// TIA Portal V17 export
// export: Created 2025-03-05T08:00:17.191262Z, ExportSetting WithDefaults, DisplayName Totally Integrated Automation Portal, DisplayVersion V17 Update 8, DisplayName TIA Portal Openness, DisplayVersion V17 Update 8, DisplayName TIA Portal Version Control Interface, DisplayVersion V17, DisplayName SINAMICS Startdrive Advanced, DisplayVersion V17 SP2, DisplayName SINAMICS Startdrive G110M, G120, G120C, G120D, G120P, G115D, DisplayVersion V17 SP2, DisplayName SINAMICS Startdrive G130, G150, S120, S150, SINAMICS MV, S210, DisplayVersion V17 SP2, DisplayName STEP 7 Professional, DisplayVersion V17 Update 8, DisplayName SINUMERIK ONE STEP 7 Toolbox, DisplayVersion V17 Update 12, DisplayName SINUMERIK 840D sl STEP 7 Toolbox, DisplayVersion V17 Update 12, DisplayName STEP 7 Safety, DisplayVersion V17 Update 6, DisplayName WinCC Advanced, DisplayVersion V17 Update 8
FUNCTION_BLOCK "FB33_SAFETY_POSITIONS"   // FB33, LAD
{ S7_Optimized_Access := 'FALSE' }
VERSION : 0.1
// stored: AutoNumber true, IsIECCheckEnabled false, SetENOAutomatically false, UDAEnableTagReadback false
   VAR_INPUT
      MEAS_SYS_1_ACTIVE_REFERENCED : Bool;   // MEASURING SYSTEM 1 ACTIVE AND REFERENCED
      MEAS_SYS_2_ACTIVE_REFERENCED : Bool;   // MEASURING SYSTEM 2 ACTIVE AND REFERENCED
      AXIS_POS : Real;   // AXIS POSITION
   END_VAR
   VAR DB_SPECIFIC
      AX_POS_0_DEGREES : Struct   // AXIS POSITION 0 DEGREES
         TOLERANCE : Real := 0.005;   // TOLERANCE
         POSITION_0_TOLERANCE_PLUS : Real;   // POSITION TOLERANCE PLUS
         POSITION_0_TOLERANCE_MINUS : Real;   // POSITION TOLERANCE MINUS
         POSITION_360_TOLERANCE_PLUS : Real;   // POSITION TOLERANCE PLUS
         POSITION_360_TOLERANCE_MINUS : Real;   // POSITION TOLERANCE MINUS
         IN_POSITION : Bool;   // AXIS POSITION 0 DEGREES
      END_STRUCT;
      AX_POS_90_DEGREES : Struct   // AXIS POSITION 90 DEGREES
         TOLERANCE : Real := 0.005;   // TOLERANCE
         POSITION_TOLERANCE_PLUS : Real;   // POSITION TOLERANCE PLUS
         POSITION_TOLERANCE_MINUS : Real;   // POSITION TOLERANCE MINUS
         IN_POSITION : Bool;   // AXIS POSITION 90 DEGREES
      END_STRUCT;
      AX_POS_180_DEGREES : Struct   // AXIS POSITION 180 DEGREES
         TOLERANCE : Real := 0.005;   // TOLERANCE
         POSITION_TOLERANCE_PLUS : Real;   // POSITION TOLERANCE PLUS
         POSITION_TOLERANCE_MINUS : Real;   // POSITION TOLERANCE MINUS
         IN_POSITION : Bool;   // AXIS POSITION 180 DEGREES
      END_STRUCT;
      AX_POS_270_DEGREES : Struct   // AXIS POSITION 270 DEGREES
         TOLERANCE : Real := 0.005;   // TOLERANCE
         POSITION_TOLERANCE_PLUS : Real;   // POSITION TOLERANCE PLUS
         POSITION_TOLERANCE_MINUS : Real;   // POSITION TOLERANCE MINUS
         IN_POSITION : Bool;   // AXIS POSITION 270 DEGREES
      END_STRUCT;
      AX_POS_MINUS_90_DEGREES : Bool;   // AXIS POSITION MINUS 90 DEGREES
      AX_POS_MINUS_180_DEGREES : Bool;   // AXIS POSITION MINUS 180 DEGREES
      AX_POS_MINUS_270_DEGREES : Bool;   // AXIS POSITION MINUS 270 DEGREES
      SAFETY_POSITION_1 : Struct   // HOME POSITION
         HMI_POSITION : Real := 1.1;   // HMI POSITION
         TOLERANCE_PLUS : Real := 0.01;   // TOLERANCE PLUS
         TOLERANCE_MINUS : Real := 0.01;   // TOLERANCE MINUS
         POSITION_TOLERANCE_PLUS : Real;   // POSITION TOLERANCE PLUS
         POSITION_TOLERANCE_MINUS : Real;   // POSITION TOLERANCE MINUS
         IN_POSITION : Bool;   // HOME POSITION
         GREATER_TOLERANCE_PLUS : Bool;   // GREATER THAN TOLERANCE PLUS
         GREATER_TOLERANCE_MINUS : Bool;   // GREATER TOLERANCE MINUS
         LOWER_TOLERANCE_PLUS : Bool;   // LOWER TOLERANCE PLUS
         LOWER_TOLERANCE_MINUS : Bool;   // LOWER TOLERANCE MINUS
      END_STRUCT;
      SAFETY_POSITION_2 : Struct   // CLEAR FIXTURE AXIS
         HMI_POSITION : Real := 1.1;   // HMI POSITION
         TOLERANCE_PLUS : Real := 0.01;   // TOLERANCE PLUS
         TOLERANCE_MINUS : Real := 0.01;   // TOLERANCE MINUS
         POSITION_TOLERANCE_PLUS : Real;   // POSITION TOLERANCE PLUS
         POSITION_TOLERANCE_MINUS : Real;   // POSITION TOLERANCE MINUS
         IN_POSITION : Bool;   // IN POSITION
         GREATER_TOLERANCE_PLUS : Bool;   // GREATER TOLERANCE PLUS
         GREATER_TOLERANCE_MINUS : Bool;   // CLEAR FIXTURE AXIS
         LOWER_TOLERANCE_PLUS : Bool;   // LOWER TOLERANCE PLUS
         LOWER_TOLERANCE_MINUS : Bool;   // LOWER TOLERANCE MINUS
      END_STRUCT;
      SAFETY_POSITION_3 : Struct   // TOOL CHANGE POSITION
         HMI_POSITION : Real := 1.1;   // HMI POSITION
         TOLERANCE_PLUS : Real := 0.01;   // TOLERANCE
         TOLERANCE_MINUS : Real := 0.01;   // TOLERANCE MINUS
         POSITION_TOLERANCE_PLUS : Real;   // POSITION TOLERANCE PLUS
         POSITION_TOLERANCE_MINUS : Real;   // POSITION TOLERANCE MINUS
         IN_POSITION : Bool;   // TOOL CHANGE POSITION
         GREATER_TOLERANCE_PLUS : Bool;   // GREATER TOLERANCE PLUS
         GREATER_TOLERANCE_MINUS : Bool;   // GREATER TOLERANCE MINUS
         LOWER_TOLERANCE_PLUS : Bool;   // LOWER TOLERANCE PLUS
         LOWER_TOLERANCE_MINUS : Bool;   // LOWER TOLERANCE MINUS
      END_STRUCT;
      SAFETY_POSITION_4 : Struct   // RETURNED
         HMI_POSITION : Real := 1.1;   // HMI POSITION
         TOLERANCE_PLUS : Real := 0.01;   // TOLERANCE PLUS
         TOLERANCE_MINUS : Real := 0.01;   // TOLERANCE MINUS
         POSITION_TOLERANCE_PLUS : Real;   // POSITION TOLERANCE PLUS
         POSITION_TOLERANCE_MINUS : Real;   // POSITION TOLERANCE MINUS
         IN_POSITION : Bool;   // RETURNED
         GREATER_TOLERANCE_PLUS : Bool;   // GREATER TOLERANCE PLUS
         GREATER_TOLERANCE_MINUS : Bool;   // GREATER TOLERANCE MINUS
         LOWER_TOLERANCE_PLUS : Bool;   // LOWER TOLERANCE PLUS
         LOWER_TOLERANCE_MINUS : Bool;   // LOWER TOLERANCE MINUS
      END_STRUCT;
      SAFETY_POSITION_5 : Struct   // ADVANCED
         HMI_POSITION : Real := 1.1;   // HMI POSITION
         TOLERANCE_PLUS : Real := 0.01;   // TOLERANCE_PLUS
         TOLERANCE_MINUS : Real := 0.01;   // TOLERANCE MINUS
         POSITION_TOLERANCE_PLUS : Real;   // POSITION TOLERANCE PLUS
         POSITION_TOLERANCE_MINUS : Real;   // POSITION TOLERANCE MINUS
         IN_POSITION : Bool;   // ADVANCED
         GREATER_TOLERANCE_PLUS : Bool;   // GREATER TOLERANCE PLUS
         GREATER_TOLERANCE_MINUS : Bool;   // GREATER TOLERANCE MINUS
         LOWER_TOLERANCE_PLUS : Bool;   // LOWER TOLERANCE PLUS
         LOWER_TOLERANCE_MINUS : Bool;   // LOWER TOLERANCE MINUS
      END_STRUCT;
      SAFETY_POSITION_6 : Struct
         HMI_POSITION : Real := 1.1;   // HMI POSITION
         TOLERANCE_PLUS : Real := 0.01;   // TOLERANCE PLUS
         TOLERANCE_MINUS : Real := 0.01;   // TOLERANCE MINUS
         POSITION_TOLERANCE_PLUS : Real;   // POSITION TOLERANCE PLUS
         POSITION_TOLERANCE_MINUS : Real;   // POSITION TOLERANCE MINUS
         IN_POSITION : Bool;   // IN POSITION
         GREATER_TOLERANCE_PLUS : Bool;   // GREATER TOLERANCE PLUS
         GREATER_TOLERANCE_MINUS : Bool;   // GREATER TOLERANCE MINUS
         LOWER_TOLERANCE_PLUS : Bool;   // LOWER TOLERANCE PLUS
         LOWER_TOLERANCE_MINUS : Bool;   // LOWER TOLERANCE MINUS
      END_STRUCT;
      SAFETY_POSITION_7 : Struct
         HMI_POSITION : Real := 1.1;   // HMI POSITION
         TOLERANCE_PLUS : Real := 0.01;   // TOLERANCE PLUS
         TOLERANCE_MINUS : Real := 0.01;   // TOLERANCE MINUS
         POSITION_TOLERANCE_PLUS : Real;   // POSITION TOLERANCE PLUS
         POSITION_TOLERANCE_MINUS : Real;   // POSITION TOLERANCE MINUS
         IN_POSITION : Bool;   // IN POSITION
         GREATER_TOLERANCE_PLUS : Bool;   // GREATER TOLERANCE PLUS
         GREATER_TOLERANCE_MINUS : Bool;   // GREATER TOLERANCE MINUS
         LOWER_TOLERANCE_PLUS : Bool;   // LOWER TOLERANCE PLUS
         LOWER_TOLERANCE_MINUS : Bool;   // LOWER TOLERANCE MINUS
      END_STRUCT;
      SAFETY_POSITION_8 : Struct
         HMI_POSITION : Real := 1.1;   // HMI POSITION
         TOLERANCE_PLUS : Real := 0.01;   // TOLERANCE PLUS
         TOLERANCE_MINUS : Real := 0.01;   // TOLERANCE MINUS
         POSITION_TOLERANCE_PLUS : Real;   // POSITION TOLERANCE PLUS
         POSITION_TOLERANCE_MINUS : Real;   // POSITION TOLERANCE MINUS
         IN_POSITION : Bool;   // IN POSITION
         GREATER_TOLERANCE_PLUS : Bool;   // GREATER TOLERANCE PLUS
         GREATER_TOLERANCE_MINUS : Bool;   // GREATER TOLERANCE MINUS
         LOWER_TOLERANCE_PLUS : Bool;   // LOWER TOLERANCE PLUS
         LOWER_TOLERANCE_MINUS : Bool;   // LOWER TOLERANCE MINUS
      END_STRUCT;
      SAFETY_POSITION_9 : Struct
         HMI_POSITION : Real := 1.1;   // HMI POSITION
         TOLERANCE_PLUS : Real := 0.01;   // TOLERANCE PLUS
         TOLERANCE_MINUS : Real := 0.01;   // TOLERANCE MINUS
         POSITION_TOLERANCE_PLUS : Real;   // POSITION TOLERANCE PLUS
         POSITION_TOLERANCE_MINUS : Real;   // POSITION TOLERANCE MINUS
         IN_POSITION : Bool;   // IN POSITION
         GREATER_TOLERANCE_PLUS : Bool;   // GREATER TOLERANCE PLUS
         GREATER_TOLERANCE_MINUS : Bool;   // GREATER TOLERANCE MINUS
         LOWER_TOLERANCE_PLUS : Bool;   // LOWER TOLERANCE PLUS
         LOWER_TOLERANCE_MINUS : Bool;   // LOWER TOLERANCE MINUS
      END_STRUCT;
      SAFETY_POSITION_10 : Struct
         HMI_POSITION : Real := 1.1;   // HMI POSITION
         TOLERANCE_PLUS : Real := 0.01;   // TOLERANCE PLUS
         TOLERANCE_MINUS : Real := 0.01;   // TOLERANCE MINUS
         POSITION_TOLERANCE_PLUS : Real;   // POSITION TOLERANCE PLUS
         POSITION_TOLERANCE_MINUS : Real;   // POSITION TOLERANCE MINUS
         IN_POSITION : Bool;   // IN POSITION
         GREATER_TOLERANCE_PLUS : Bool;   // GREATER TOLERANCE PLUS
         GREATER_TOLERANCE_MINUS : Bool;   // GREATER TOLERANCE MINUS
         LOWER_TOLERANCE_PLUS : Bool;   // LOWER TOLERANCE PLUS
         LOWER_TOLERANCE_MINUS : Bool;   // LOWER TOLERANCE MINUS
      END_STRUCT;
   END_VAR
   VAR_TEMP   // added for the SCL form of the ladder/FBD networks
      _w1 : Bool;
      _w2 : Bool;
   END_VAR
BEGIN

REGION Network 1: AXIS POSITION 0 DEGREES
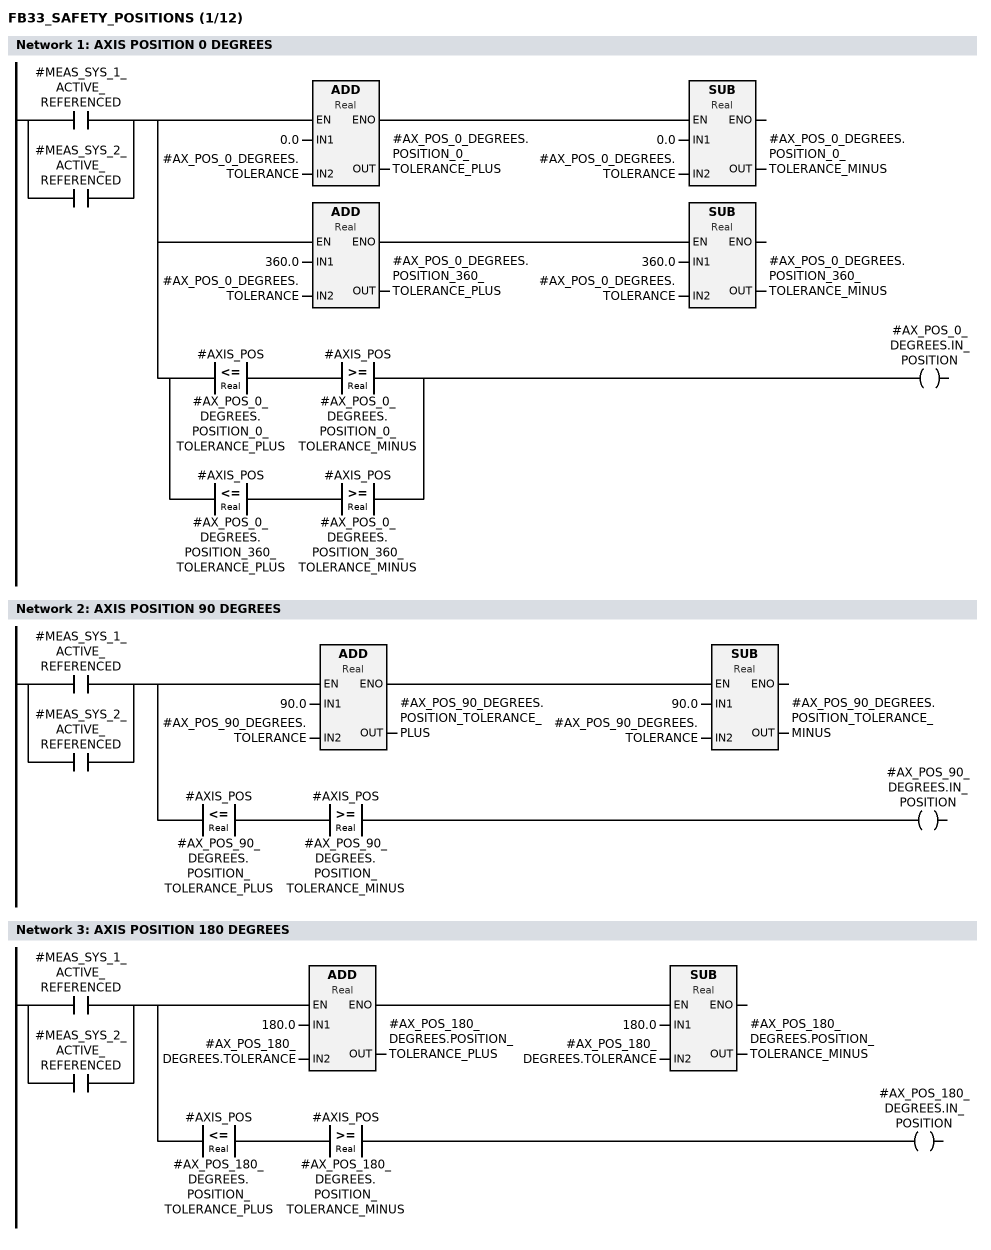
   RUNG wire#powerrail
      Contact( #MEAS_SYS_1_ACTIVE_REFERENCED )
      wire#w1
      { S7_Templates := "SrcType := Real"; S7_GenerateENO := "TRUE" } Add(in1 := 0.0, in2 := #AX_POS_0_DEGREES.TOLERANCE, out => #AX_POS_0_DEGREES.POSITION_0_TOLERANCE_PLUS)
      { S7_Templates := "SrcType := Real"; S7_GenerateENO := "TRUE" } Sub(in1 := 0.0, in2 := #AX_POS_0_DEGREES.TOLERANCE, out => #AX_POS_0_DEGREES.POSITION_0_TOLERANCE_MINUS)
   END_RUNG
   RUNG wire#powerrail
      Contact( #MEAS_SYS_2_ACTIVE_REFERENCED )
   END_RUNG wire#w1
   RUNG wire#w1
      { S7_Templates := "SrcType := Real"; S7_GenerateENO := "TRUE" } Add(in1 := 360.0, in2 := #AX_POS_0_DEGREES.TOLERANCE, out => #AX_POS_0_DEGREES.POSITION_360_TOLERANCE_PLUS)
      { S7_Templates := "SrcType := Real"; S7_GenerateENO := "TRUE" } Sub(in1 := 360.0, in2 := #AX_POS_0_DEGREES.TOLERANCE, out => #AX_POS_0_DEGREES.POSITION_360_TOLERANCE_MINUS)
   END_RUNG
   RUNG wire#w1
      { S7_Templates := "SrcType := Real" } LE_Contact(in1 := #AXIS_POS, in2 := #AX_POS_0_DEGREES.POSITION_0_TOLERANCE_PLUS)
      { S7_Templates := "SrcType := Real" } GE_Contact(in1 := #AXIS_POS, in2 := #AX_POS_0_DEGREES.POSITION_0_TOLERANCE_MINUS)
      wire#w2
      Coil( #AX_POS_0_DEGREES.IN_POSITION )
   END_RUNG
   RUNG wire#w1
      { S7_Templates := "SrcType := Real" } LE_Contact(in1 := #AXIS_POS, in2 := #AX_POS_0_DEGREES.POSITION_360_TOLERANCE_PLUS)
      { S7_Templates := "SrcType := Real" } GE_Contact(in1 := #AXIS_POS, in2 := #AX_POS_0_DEGREES.POSITION_360_TOLERANCE_MINUS)
   END_RUNG wire#w2
   // the same network as SCL:
   // ENO of a box is taken as its EN; it also drops when the box reports an error
   #_w1 := #MEAS_SYS_1_ACTIVE_REFERENCED OR #MEAS_SYS_2_ACTIVE_REFERENCED;
   IF #_w1 THEN
       #AX_POS_0_DEGREES.POSITION_0_TOLERANCE_PLUS := 0.0 + #AX_POS_0_DEGREES.TOLERANCE;
       #AX_POS_0_DEGREES.POSITION_0_TOLERANCE_MINUS := 0.0 - #AX_POS_0_DEGREES.TOLERANCE;
       #AX_POS_0_DEGREES.POSITION_360_TOLERANCE_PLUS := 360.0 + #AX_POS_0_DEGREES.TOLERANCE;
       #AX_POS_0_DEGREES.POSITION_360_TOLERANCE_MINUS := 360.0 - #AX_POS_0_DEGREES.TOLERANCE;
   END_IF;
   #AX_POS_0_DEGREES.IN_POSITION := #_w1 AND (((#AXIS_POS <= #AX_POS_0_DEGREES.POSITION_0_TOLERANCE_PLUS) AND (#AXIS_POS >= #AX_POS_0_DEGREES.POSITION_0_TOLERANCE_MINUS)) OR ((#AXIS_POS <= #AX_POS_0_DEGREES.POSITION_360_TOLERANCE_PLUS) AND (#AXIS_POS >= #AX_POS_0_DEGREES.POSITION_360_TOLERANCE_MINUS)));
END_REGION

REGION Network 2: AXIS POSITION 90 DEGREES
   RUNG wire#powerrail
      Contact( #MEAS_SYS_1_ACTIVE_REFERENCED )
      wire#w1
      { S7_Templates := "SrcType := Real"; S7_GenerateENO := "TRUE" } Add(in1 := 90.0, in2 := #AX_POS_90_DEGREES.TOLERANCE, out => #AX_POS_90_DEGREES.POSITION_TOLERANCE_PLUS)
      { S7_Templates := "SrcType := Real"; S7_GenerateENO := "TRUE" } Sub(in1 := 90.0, in2 := #AX_POS_90_DEGREES.TOLERANCE, out => #AX_POS_90_DEGREES.POSITION_TOLERANCE_MINUS)
   END_RUNG
   RUNG wire#powerrail
      Contact( #MEAS_SYS_2_ACTIVE_REFERENCED )
   END_RUNG wire#w1
   RUNG wire#w1
      { S7_Templates := "SrcType := Real" } LE_Contact(in1 := #AXIS_POS, in2 := #AX_POS_90_DEGREES.POSITION_TOLERANCE_PLUS)
      { S7_Templates := "SrcType := Real" } GE_Contact(in1 := #AXIS_POS, in2 := #AX_POS_90_DEGREES.POSITION_TOLERANCE_MINUS)
      Coil( #AX_POS_90_DEGREES.IN_POSITION )
   END_RUNG
   // the same network as SCL:
   // ENO of a box is taken as its EN; it also drops when the box reports an error
   #_w1 := #MEAS_SYS_1_ACTIVE_REFERENCED OR #MEAS_SYS_2_ACTIVE_REFERENCED;
   IF #_w1 THEN
       #AX_POS_90_DEGREES.POSITION_TOLERANCE_PLUS := 90.0 + #AX_POS_90_DEGREES.TOLERANCE;
       #AX_POS_90_DEGREES.POSITION_TOLERANCE_MINUS := 90.0 - #AX_POS_90_DEGREES.TOLERANCE;
   END_IF;
   #AX_POS_90_DEGREES.IN_POSITION := #_w1 AND (#AXIS_POS <= #AX_POS_90_DEGREES.POSITION_TOLERANCE_PLUS) AND (#AXIS_POS >= #AX_POS_90_DEGREES.POSITION_TOLERANCE_MINUS);
END_REGION

REGION Network 3: AXIS POSITION 180 DEGREES
   RUNG wire#powerrail
      Contact( #MEAS_SYS_1_ACTIVE_REFERENCED )
      wire#w1
      { S7_Templates := "SrcType := Real"; S7_GenerateENO := "TRUE" } Add(in1 := 180.0, in2 := #AX_POS_180_DEGREES.TOLERANCE, out => #AX_POS_180_DEGREES.POSITION_TOLERANCE_PLUS)
      { S7_Templates := "SrcType := Real"; S7_GenerateENO := "TRUE" } Sub(in1 := 180.0, in2 := #AX_POS_180_DEGREES.TOLERANCE, out => #AX_POS_180_DEGREES.POSITION_TOLERANCE_MINUS)
   END_RUNG
   RUNG wire#powerrail
      Contact( #MEAS_SYS_2_ACTIVE_REFERENCED )
   END_RUNG wire#w1
   RUNG wire#w1
      { S7_Templates := "SrcType := Real" } LE_Contact(in1 := #AXIS_POS, in2 := #AX_POS_180_DEGREES.POSITION_TOLERANCE_PLUS)
      { S7_Templates := "SrcType := Real" } GE_Contact(in1 := #AXIS_POS, in2 := #AX_POS_180_DEGREES.POSITION_TOLERANCE_MINUS)
      Coil( #AX_POS_180_DEGREES.IN_POSITION )
   END_RUNG
   // the same network as SCL:
   // ENO of a box is taken as its EN; it also drops when the box reports an error
   #_w1 := #MEAS_SYS_1_ACTIVE_REFERENCED OR #MEAS_SYS_2_ACTIVE_REFERENCED;
   IF #_w1 THEN
       #AX_POS_180_DEGREES.POSITION_TOLERANCE_PLUS := 180.0 + #AX_POS_180_DEGREES.TOLERANCE;
       #AX_POS_180_DEGREES.POSITION_TOLERANCE_MINUS := 180.0 - #AX_POS_180_DEGREES.TOLERANCE;
   END_IF;
   #AX_POS_180_DEGREES.IN_POSITION := #_w1 AND (#AXIS_POS <= #AX_POS_180_DEGREES.POSITION_TOLERANCE_PLUS) AND (#AXIS_POS >= #AX_POS_180_DEGREES.POSITION_TOLERANCE_MINUS);
END_REGION

REGION Network 4: AXIS POSITION 270 DEGREES
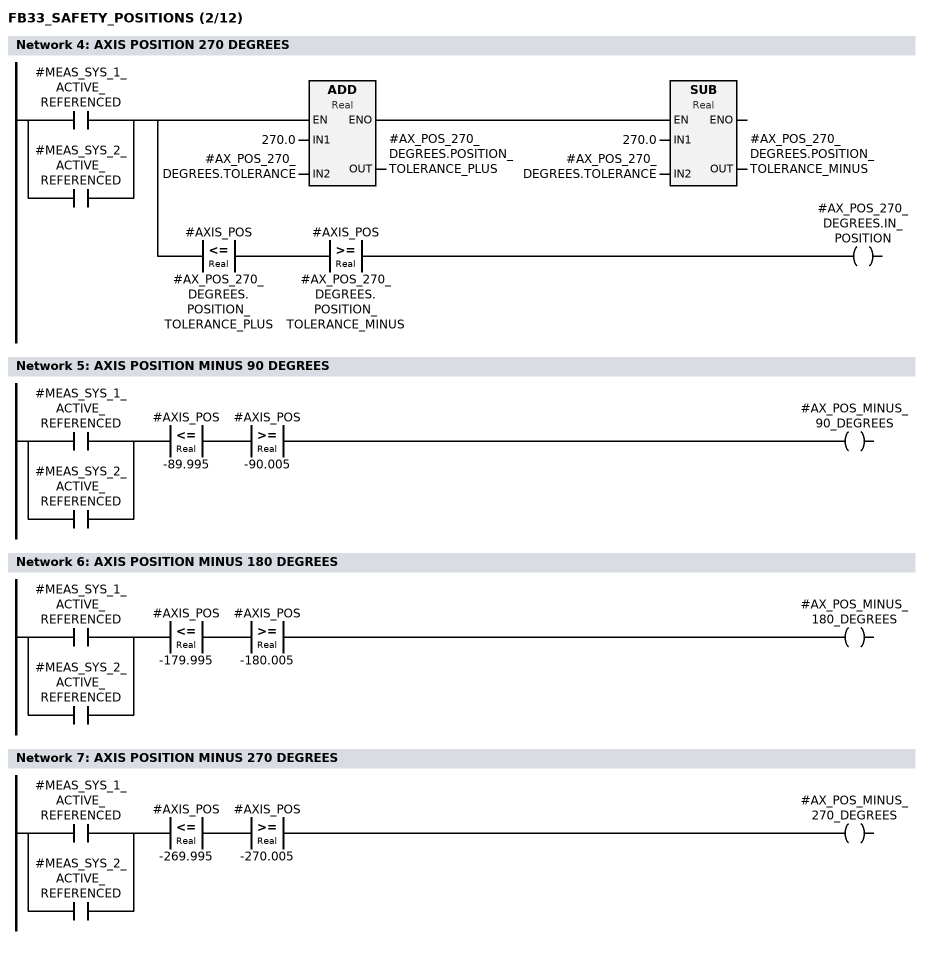
   RUNG wire#powerrail
      Contact( #MEAS_SYS_1_ACTIVE_REFERENCED )
      wire#w1
      { S7_Templates := "SrcType := Real"; S7_GenerateENO := "TRUE" } Add(in1 := 270.0, in2 := #AX_POS_270_DEGREES.TOLERANCE, out => #AX_POS_270_DEGREES.POSITION_TOLERANCE_PLUS)
      { S7_Templates := "SrcType := Real"; S7_GenerateENO := "TRUE" } Sub(in1 := 270.0, in2 := #AX_POS_270_DEGREES.TOLERANCE, out => #AX_POS_270_DEGREES.POSITION_TOLERANCE_MINUS)
   END_RUNG
   RUNG wire#powerrail
      Contact( #MEAS_SYS_2_ACTIVE_REFERENCED )
   END_RUNG wire#w1
   RUNG wire#w1
      { S7_Templates := "SrcType := Real" } LE_Contact(in1 := #AXIS_POS, in2 := #AX_POS_270_DEGREES.POSITION_TOLERANCE_PLUS)
      { S7_Templates := "SrcType := Real" } GE_Contact(in1 := #AXIS_POS, in2 := #AX_POS_270_DEGREES.POSITION_TOLERANCE_MINUS)
      Coil( #AX_POS_270_DEGREES.IN_POSITION )
   END_RUNG
   // the same network as SCL:
   // ENO of a box is taken as its EN; it also drops when the box reports an error
   #_w1 := #MEAS_SYS_1_ACTIVE_REFERENCED OR #MEAS_SYS_2_ACTIVE_REFERENCED;
   IF #_w1 THEN
       #AX_POS_270_DEGREES.POSITION_TOLERANCE_PLUS := 270.0 + #AX_POS_270_DEGREES.TOLERANCE;
       #AX_POS_270_DEGREES.POSITION_TOLERANCE_MINUS := 270.0 - #AX_POS_270_DEGREES.TOLERANCE;
   END_IF;
   #AX_POS_270_DEGREES.IN_POSITION := #_w1 AND (#AXIS_POS <= #AX_POS_270_DEGREES.POSITION_TOLERANCE_PLUS) AND (#AXIS_POS >= #AX_POS_270_DEGREES.POSITION_TOLERANCE_MINUS);
END_REGION

REGION Network 5: AXIS POSITION MINUS 90 DEGREES
   RUNG wire#powerrail
      Contact( #MEAS_SYS_1_ACTIVE_REFERENCED )
      wire#w1
      { S7_Templates := "SrcType := Real" } LE_Contact(in1 := #AXIS_POS, in2 := -89.995)
      { S7_Templates := "SrcType := Real" } GE_Contact(in1 := #AXIS_POS, in2 := -90.005)
      Coil( #AX_POS_MINUS_90_DEGREES )
   END_RUNG
   RUNG wire#powerrail
      Contact( #MEAS_SYS_2_ACTIVE_REFERENCED )
   END_RUNG wire#w1
   // the same network as SCL:
   #AX_POS_MINUS_90_DEGREES := (#MEAS_SYS_1_ACTIVE_REFERENCED OR #MEAS_SYS_2_ACTIVE_REFERENCED) AND (#AXIS_POS <= (-89.995)) AND (#AXIS_POS >= (-90.005));
END_REGION

REGION Network 6: AXIS POSITION MINUS 180 DEGREES
   RUNG wire#powerrail
      Contact( #MEAS_SYS_1_ACTIVE_REFERENCED )
      wire#w1
      { S7_Templates := "SrcType := Real" } LE_Contact(in1 := #AXIS_POS, in2 := -179.995)
      { S7_Templates := "SrcType := Real" } GE_Contact(in1 := #AXIS_POS, in2 := -180.005)
      Coil( #AX_POS_MINUS_180_DEGREES )
   END_RUNG
   RUNG wire#powerrail
      Contact( #MEAS_SYS_2_ACTIVE_REFERENCED )
   END_RUNG wire#w1
   // the same network as SCL:
   #AX_POS_MINUS_180_DEGREES := (#MEAS_SYS_1_ACTIVE_REFERENCED OR #MEAS_SYS_2_ACTIVE_REFERENCED) AND (#AXIS_POS <= (-179.995)) AND (#AXIS_POS >= (-180.005));
END_REGION

REGION Network 7: AXIS POSITION MINUS 270 DEGREES
   RUNG wire#powerrail
      Contact( #MEAS_SYS_1_ACTIVE_REFERENCED )
      wire#w1
      { S7_Templates := "SrcType := Real" } LE_Contact(in1 := #AXIS_POS, in2 := -269.995)
      { S7_Templates := "SrcType := Real" } GE_Contact(in1 := #AXIS_POS, in2 := -270.005)
      Coil( #AX_POS_MINUS_270_DEGREES )
   END_RUNG
   RUNG wire#powerrail
      Contact( #MEAS_SYS_2_ACTIVE_REFERENCED )
   END_RUNG wire#w1
   // the same network as SCL:
   #AX_POS_MINUS_270_DEGREES := (#MEAS_SYS_1_ACTIVE_REFERENCED OR #MEAS_SYS_2_ACTIVE_REFERENCED) AND (#AXIS_POS <= (-269.995)) AND (#AXIS_POS >= (-270.005));
END_REGION

REGION Network 8: SAFETY POSITION 1
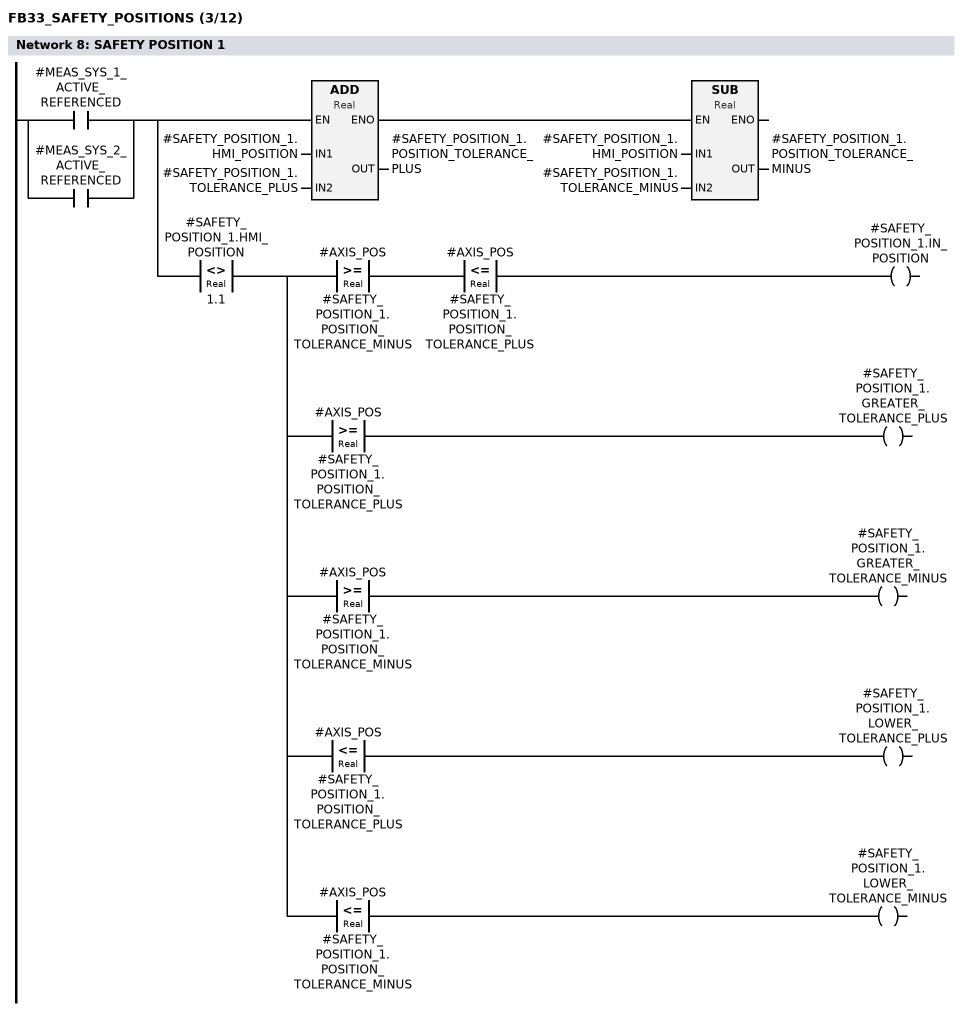
   RUNG wire#powerrail
      Contact( #MEAS_SYS_1_ACTIVE_REFERENCED )
      wire#w1
      { S7_Templates := "SrcType := Real"; S7_GenerateENO := "TRUE" } Add(in1 := #SAFETY_POSITION_1.HMI_POSITION, in2 := #SAFETY_POSITION_1.TOLERANCE_PLUS, out => #SAFETY_POSITION_1.POSITION_TOLERANCE_PLUS)
      { S7_Templates := "SrcType := Real"; S7_GenerateENO := "TRUE" } Sub(in1 := #SAFETY_POSITION_1.HMI_POSITION, in2 := #SAFETY_POSITION_1.TOLERANCE_MINUS, out => #SAFETY_POSITION_1.POSITION_TOLERANCE_MINUS)
   END_RUNG
   RUNG wire#powerrail
      Contact( #MEAS_SYS_2_ACTIVE_REFERENCED )
   END_RUNG wire#w1
   RUNG wire#w1
      { S7_Templates := "SrcType := Real" } NE_Contact(in1 := #SAFETY_POSITION_1.HMI_POSITION, in2 := 1.1)
      wire#w2
      { S7_Templates := "SrcType := Real" } GE_Contact(in1 := #AXIS_POS, in2 := #SAFETY_POSITION_1.POSITION_TOLERANCE_MINUS)
      { S7_Templates := "SrcType := Real" } LE_Contact(in1 := #AXIS_POS, in2 := #SAFETY_POSITION_1.POSITION_TOLERANCE_PLUS)
      Coil( #SAFETY_POSITION_1.IN_POSITION )
   END_RUNG
   RUNG wire#w2
      { S7_Templates := "SrcType := Real" } GE_Contact(in1 := #AXIS_POS, in2 := #SAFETY_POSITION_1.POSITION_TOLERANCE_PLUS)
      Coil( #SAFETY_POSITION_1.GREATER_TOLERANCE_PLUS )
   END_RUNG
   RUNG wire#w2
      { S7_Templates := "SrcType := Real" } GE_Contact(in1 := #AXIS_POS, in2 := #SAFETY_POSITION_1.POSITION_TOLERANCE_MINUS)
      Coil( #SAFETY_POSITION_1.GREATER_TOLERANCE_MINUS )
   END_RUNG
   RUNG wire#w2
      { S7_Templates := "SrcType := Real" } LE_Contact(in1 := #AXIS_POS, in2 := #SAFETY_POSITION_1.POSITION_TOLERANCE_PLUS)
      Coil( #SAFETY_POSITION_1.LOWER_TOLERANCE_PLUS )
   END_RUNG
   RUNG wire#w2
      { S7_Templates := "SrcType := Real" } LE_Contact(in1 := #AXIS_POS, in2 := #SAFETY_POSITION_1.POSITION_TOLERANCE_MINUS)
      Coil( #SAFETY_POSITION_1.LOWER_TOLERANCE_MINUS )
   END_RUNG
   // the same network as SCL:
   // ENO of a box is taken as its EN; it also drops when the box reports an error
   #_w1 := #MEAS_SYS_1_ACTIVE_REFERENCED OR #MEAS_SYS_2_ACTIVE_REFERENCED;
   IF #_w1 THEN
       #SAFETY_POSITION_1.POSITION_TOLERANCE_PLUS := #SAFETY_POSITION_1.HMI_POSITION + #SAFETY_POSITION_1.TOLERANCE_PLUS;
       #SAFETY_POSITION_1.POSITION_TOLERANCE_MINUS := #SAFETY_POSITION_1.HMI_POSITION - #SAFETY_POSITION_1.TOLERANCE_MINUS;
   END_IF;
   #_w2 := #_w1 AND (#SAFETY_POSITION_1.HMI_POSITION <> 1.1);
   #SAFETY_POSITION_1.IN_POSITION := #_w2 AND (#AXIS_POS >= #SAFETY_POSITION_1.POSITION_TOLERANCE_MINUS) AND (#AXIS_POS <= #SAFETY_POSITION_1.POSITION_TOLERANCE_PLUS);
   #SAFETY_POSITION_1.GREATER_TOLERANCE_PLUS := #_w2 AND (#AXIS_POS >= #SAFETY_POSITION_1.POSITION_TOLERANCE_PLUS);
   #SAFETY_POSITION_1.GREATER_TOLERANCE_MINUS := #_w2 AND (#AXIS_POS >= #SAFETY_POSITION_1.POSITION_TOLERANCE_MINUS);
   #SAFETY_POSITION_1.LOWER_TOLERANCE_PLUS := #_w2 AND (#AXIS_POS <= #SAFETY_POSITION_1.POSITION_TOLERANCE_PLUS);
   #SAFETY_POSITION_1.LOWER_TOLERANCE_MINUS := #_w2 AND (#AXIS_POS <= #SAFETY_POSITION_1.POSITION_TOLERANCE_MINUS);
END_REGION

REGION Network 9: SAFETY POSITION 2
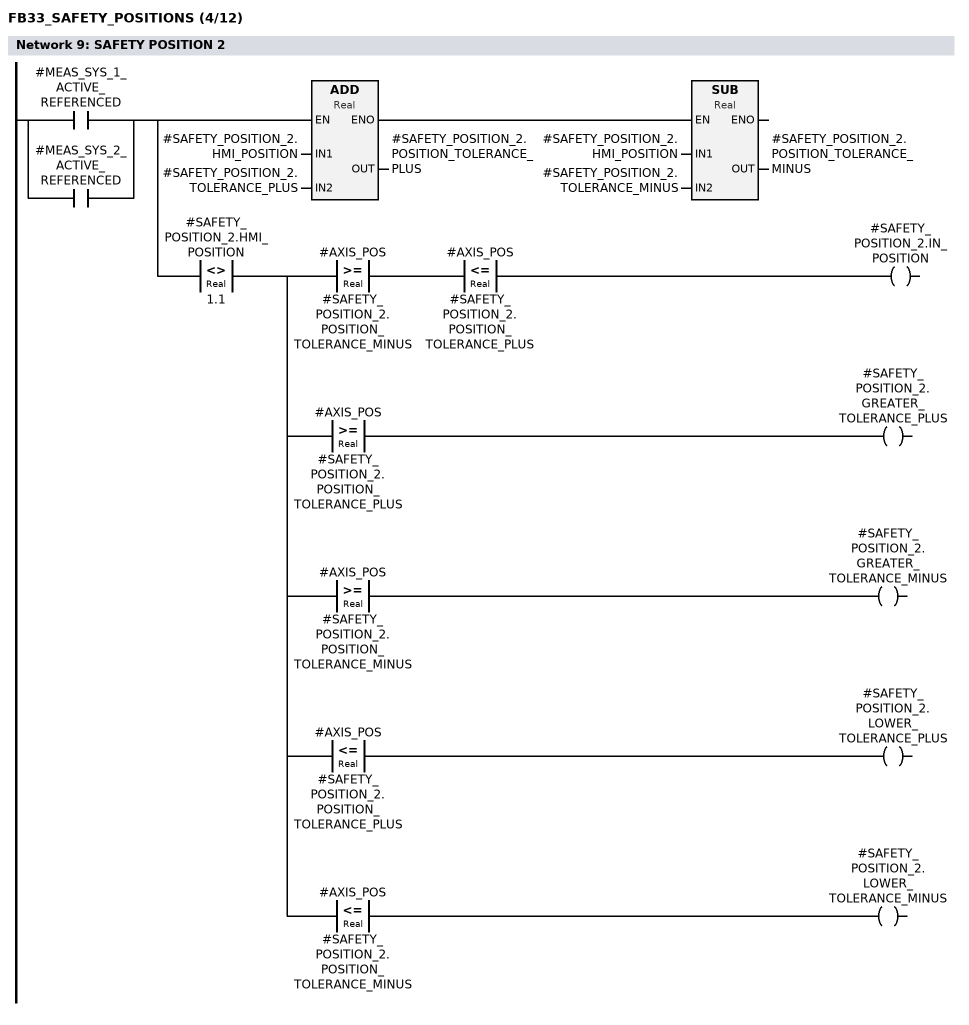
   RUNG wire#powerrail
      Contact( #MEAS_SYS_1_ACTIVE_REFERENCED )
      wire#w1
      { S7_Templates := "SrcType := Real"; S7_GenerateENO := "TRUE" } Add(in1 := #SAFETY_POSITION_2.HMI_POSITION, in2 := #SAFETY_POSITION_2.TOLERANCE_PLUS, out => #SAFETY_POSITION_2.POSITION_TOLERANCE_PLUS)
      { S7_Templates := "SrcType := Real"; S7_GenerateENO := "TRUE" } Sub(in1 := #SAFETY_POSITION_2.HMI_POSITION, in2 := #SAFETY_POSITION_2.TOLERANCE_MINUS, out => #SAFETY_POSITION_2.POSITION_TOLERANCE_MINUS)
   END_RUNG
   RUNG wire#powerrail
      Contact( #MEAS_SYS_2_ACTIVE_REFERENCED )
   END_RUNG wire#w1
   RUNG wire#w1
      { S7_Templates := "SrcType := Real" } NE_Contact(in1 := #SAFETY_POSITION_2.HMI_POSITION, in2 := 1.1)
      wire#w2
      { S7_Templates := "SrcType := Real" } GE_Contact(in1 := #AXIS_POS, in2 := #SAFETY_POSITION_2.POSITION_TOLERANCE_MINUS)
      { S7_Templates := "SrcType := Real" } LE_Contact(in1 := #AXIS_POS, in2 := #SAFETY_POSITION_2.POSITION_TOLERANCE_PLUS)
      Coil( #SAFETY_POSITION_2.IN_POSITION )
   END_RUNG
   RUNG wire#w2
      { S7_Templates := "SrcType := Real" } GE_Contact(in1 := #AXIS_POS, in2 := #SAFETY_POSITION_2.POSITION_TOLERANCE_PLUS)
      Coil( #SAFETY_POSITION_2.GREATER_TOLERANCE_PLUS )
   END_RUNG
   RUNG wire#w2
      { S7_Templates := "SrcType := Real" } GE_Contact(in1 := #AXIS_POS, in2 := #SAFETY_POSITION_2.POSITION_TOLERANCE_MINUS)
      Coil( #SAFETY_POSITION_2.GREATER_TOLERANCE_MINUS )
   END_RUNG
   RUNG wire#w2
      { S7_Templates := "SrcType := Real" } LE_Contact(in1 := #AXIS_POS, in2 := #SAFETY_POSITION_2.POSITION_TOLERANCE_PLUS)
      Coil( #SAFETY_POSITION_2.LOWER_TOLERANCE_PLUS )
   END_RUNG
   RUNG wire#w2
      { S7_Templates := "SrcType := Real" } LE_Contact(in1 := #AXIS_POS, in2 := #SAFETY_POSITION_2.POSITION_TOLERANCE_MINUS)
      Coil( #SAFETY_POSITION_2.LOWER_TOLERANCE_MINUS )
   END_RUNG
   // the same network as SCL:
   // ENO of a box is taken as its EN; it also drops when the box reports an error
   #_w1 := #MEAS_SYS_1_ACTIVE_REFERENCED OR #MEAS_SYS_2_ACTIVE_REFERENCED;
   IF #_w1 THEN
       #SAFETY_POSITION_2.POSITION_TOLERANCE_PLUS := #SAFETY_POSITION_2.HMI_POSITION + #SAFETY_POSITION_2.TOLERANCE_PLUS;
       #SAFETY_POSITION_2.POSITION_TOLERANCE_MINUS := #SAFETY_POSITION_2.HMI_POSITION - #SAFETY_POSITION_2.TOLERANCE_MINUS;
   END_IF;
   #_w2 := #_w1 AND (#SAFETY_POSITION_2.HMI_POSITION <> 1.1);
   #SAFETY_POSITION_2.IN_POSITION := #_w2 AND (#AXIS_POS >= #SAFETY_POSITION_2.POSITION_TOLERANCE_MINUS) AND (#AXIS_POS <= #SAFETY_POSITION_2.POSITION_TOLERANCE_PLUS);
   #SAFETY_POSITION_2.GREATER_TOLERANCE_PLUS := #_w2 AND (#AXIS_POS >= #SAFETY_POSITION_2.POSITION_TOLERANCE_PLUS);
   #SAFETY_POSITION_2.GREATER_TOLERANCE_MINUS := #_w2 AND (#AXIS_POS >= #SAFETY_POSITION_2.POSITION_TOLERANCE_MINUS);
   #SAFETY_POSITION_2.LOWER_TOLERANCE_PLUS := #_w2 AND (#AXIS_POS <= #SAFETY_POSITION_2.POSITION_TOLERANCE_PLUS);
   #SAFETY_POSITION_2.LOWER_TOLERANCE_MINUS := #_w2 AND (#AXIS_POS <= #SAFETY_POSITION_2.POSITION_TOLERANCE_MINUS);
END_REGION

REGION Network 10: SAFETY POSITION 3
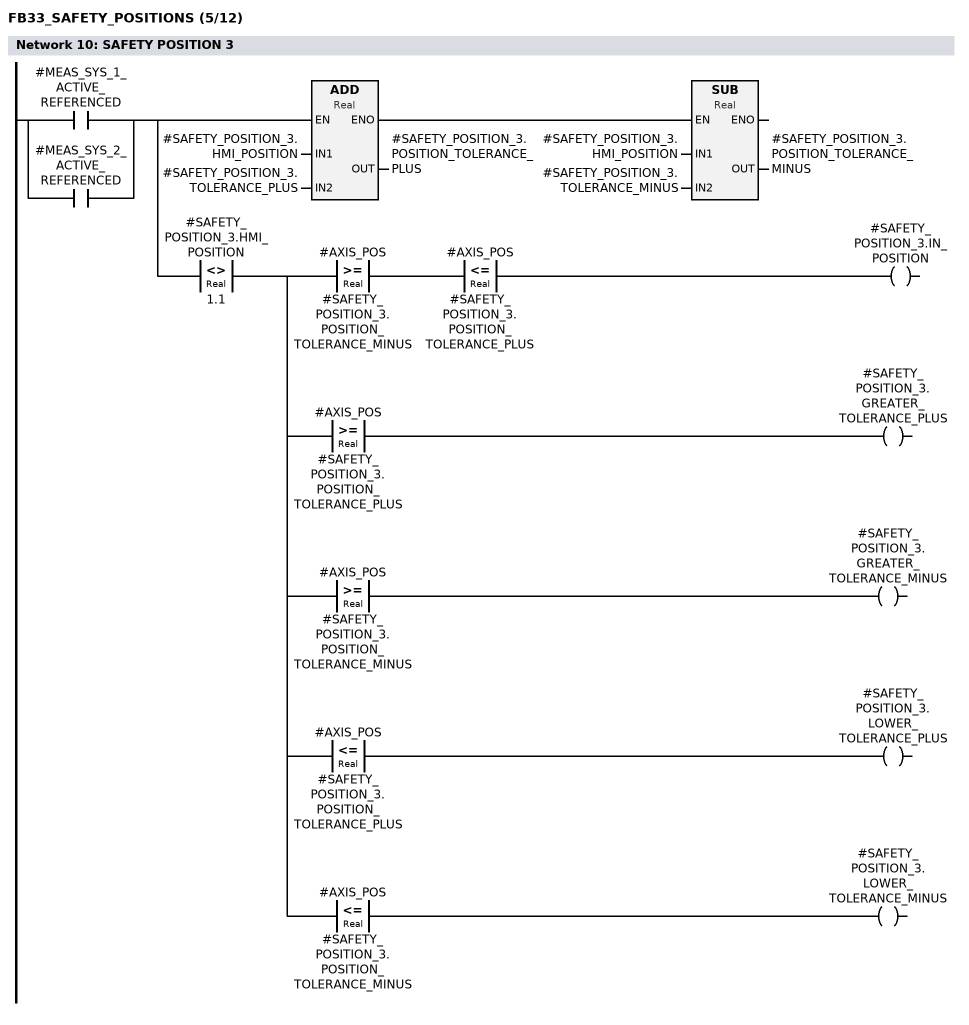
   RUNG wire#powerrail
      Contact( #MEAS_SYS_1_ACTIVE_REFERENCED )
      wire#w1
      { S7_Templates := "SrcType := Real"; S7_GenerateENO := "TRUE" } Add(in1 := #SAFETY_POSITION_3.HMI_POSITION, in2 := #SAFETY_POSITION_3.TOLERANCE_PLUS, out => #SAFETY_POSITION_3.POSITION_TOLERANCE_PLUS)
      { S7_Templates := "SrcType := Real"; S7_GenerateENO := "TRUE" } Sub(in1 := #SAFETY_POSITION_3.HMI_POSITION, in2 := #SAFETY_POSITION_3.TOLERANCE_MINUS, out => #SAFETY_POSITION_3.POSITION_TOLERANCE_MINUS)
   END_RUNG
   RUNG wire#powerrail
      Contact( #MEAS_SYS_2_ACTIVE_REFERENCED )
   END_RUNG wire#w1
   RUNG wire#w1
      { S7_Templates := "SrcType := Real" } NE_Contact(in1 := #SAFETY_POSITION_3.HMI_POSITION, in2 := 1.1)
      wire#w2
      { S7_Templates := "SrcType := Real" } GE_Contact(in1 := #AXIS_POS, in2 := #SAFETY_POSITION_3.POSITION_TOLERANCE_MINUS)
      { S7_Templates := "SrcType := Real" } LE_Contact(in1 := #AXIS_POS, in2 := #SAFETY_POSITION_3.POSITION_TOLERANCE_PLUS)
      Coil( #SAFETY_POSITION_3.IN_POSITION )
   END_RUNG
   RUNG wire#w2
      { S7_Templates := "SrcType := Real" } GE_Contact(in1 := #AXIS_POS, in2 := #SAFETY_POSITION_3.POSITION_TOLERANCE_PLUS)
      Coil( #SAFETY_POSITION_3.GREATER_TOLERANCE_PLUS )
   END_RUNG
   RUNG wire#w2
      { S7_Templates := "SrcType := Real" } GE_Contact(in1 := #AXIS_POS, in2 := #SAFETY_POSITION_3.POSITION_TOLERANCE_MINUS)
      Coil( #SAFETY_POSITION_3.GREATER_TOLERANCE_MINUS )
   END_RUNG
   RUNG wire#w2
      { S7_Templates := "SrcType := Real" } LE_Contact(in1 := #AXIS_POS, in2 := #SAFETY_POSITION_3.POSITION_TOLERANCE_PLUS)
      Coil( #SAFETY_POSITION_3.LOWER_TOLERANCE_PLUS )
   END_RUNG
   RUNG wire#w2
      { S7_Templates := "SrcType := Real" } LE_Contact(in1 := #AXIS_POS, in2 := #SAFETY_POSITION_3.POSITION_TOLERANCE_MINUS)
      Coil( #SAFETY_POSITION_3.LOWER_TOLERANCE_MINUS )
   END_RUNG
   // the same network as SCL:
   // ENO of a box is taken as its EN; it also drops when the box reports an error
   #_w1 := #MEAS_SYS_1_ACTIVE_REFERENCED OR #MEAS_SYS_2_ACTIVE_REFERENCED;
   IF #_w1 THEN
       #SAFETY_POSITION_3.POSITION_TOLERANCE_PLUS := #SAFETY_POSITION_3.HMI_POSITION + #SAFETY_POSITION_3.TOLERANCE_PLUS;
       #SAFETY_POSITION_3.POSITION_TOLERANCE_MINUS := #SAFETY_POSITION_3.HMI_POSITION - #SAFETY_POSITION_3.TOLERANCE_MINUS;
   END_IF;
   #_w2 := #_w1 AND (#SAFETY_POSITION_3.HMI_POSITION <> 1.1);
   #SAFETY_POSITION_3.IN_POSITION := #_w2 AND (#AXIS_POS >= #SAFETY_POSITION_3.POSITION_TOLERANCE_MINUS) AND (#AXIS_POS <= #SAFETY_POSITION_3.POSITION_TOLERANCE_PLUS);
   #SAFETY_POSITION_3.GREATER_TOLERANCE_PLUS := #_w2 AND (#AXIS_POS >= #SAFETY_POSITION_3.POSITION_TOLERANCE_PLUS);
   #SAFETY_POSITION_3.GREATER_TOLERANCE_MINUS := #_w2 AND (#AXIS_POS >= #SAFETY_POSITION_3.POSITION_TOLERANCE_MINUS);
   #SAFETY_POSITION_3.LOWER_TOLERANCE_PLUS := #_w2 AND (#AXIS_POS <= #SAFETY_POSITION_3.POSITION_TOLERANCE_PLUS);
   #SAFETY_POSITION_3.LOWER_TOLERANCE_MINUS := #_w2 AND (#AXIS_POS <= #SAFETY_POSITION_3.POSITION_TOLERANCE_MINUS);
END_REGION

REGION Network 11: SAFETY POSITION 4
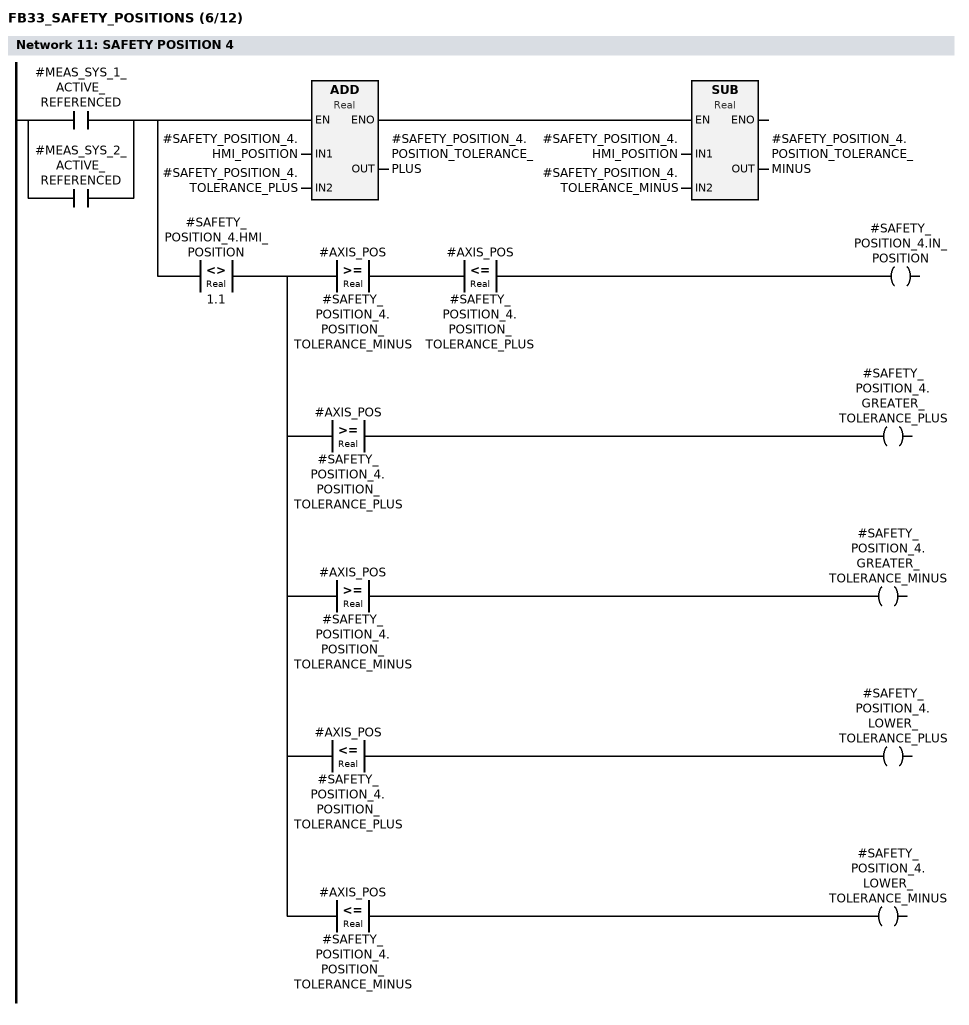
   RUNG wire#powerrail
      Contact( #MEAS_SYS_1_ACTIVE_REFERENCED )
      wire#w1
      { S7_Templates := "SrcType := Real"; S7_GenerateENO := "TRUE" } Add(in1 := #SAFETY_POSITION_4.HMI_POSITION, in2 := #SAFETY_POSITION_4.TOLERANCE_PLUS, out => #SAFETY_POSITION_4.POSITION_TOLERANCE_PLUS)
      { S7_Templates := "SrcType := Real"; S7_GenerateENO := "TRUE" } Sub(in1 := #SAFETY_POSITION_4.HMI_POSITION, in2 := #SAFETY_POSITION_4.TOLERANCE_MINUS, out => #SAFETY_POSITION_4.POSITION_TOLERANCE_MINUS)
   END_RUNG
   RUNG wire#powerrail
      Contact( #MEAS_SYS_2_ACTIVE_REFERENCED )
   END_RUNG wire#w1
   RUNG wire#w1
      { S7_Templates := "SrcType := Real" } NE_Contact(in1 := #SAFETY_POSITION_4.HMI_POSITION, in2 := 1.1)
      wire#w2
      { S7_Templates := "SrcType := Real" } GE_Contact(in1 := #AXIS_POS, in2 := #SAFETY_POSITION_4.POSITION_TOLERANCE_MINUS)
      { S7_Templates := "SrcType := Real" } LE_Contact(in1 := #AXIS_POS, in2 := #SAFETY_POSITION_4.POSITION_TOLERANCE_PLUS)
      Coil( #SAFETY_POSITION_4.IN_POSITION )
   END_RUNG
   RUNG wire#w2
      { S7_Templates := "SrcType := Real" } GE_Contact(in1 := #AXIS_POS, in2 := #SAFETY_POSITION_4.POSITION_TOLERANCE_PLUS)
      Coil( #SAFETY_POSITION_4.GREATER_TOLERANCE_PLUS )
   END_RUNG
   RUNG wire#w2
      { S7_Templates := "SrcType := Real" } GE_Contact(in1 := #AXIS_POS, in2 := #SAFETY_POSITION_4.POSITION_TOLERANCE_MINUS)
      Coil( #SAFETY_POSITION_4.GREATER_TOLERANCE_MINUS )
   END_RUNG
   RUNG wire#w2
      { S7_Templates := "SrcType := Real" } LE_Contact(in1 := #AXIS_POS, in2 := #SAFETY_POSITION_4.POSITION_TOLERANCE_PLUS)
      Coil( #SAFETY_POSITION_4.LOWER_TOLERANCE_PLUS )
   END_RUNG
   RUNG wire#w2
      { S7_Templates := "SrcType := Real" } LE_Contact(in1 := #AXIS_POS, in2 := #SAFETY_POSITION_4.POSITION_TOLERANCE_MINUS)
      Coil( #SAFETY_POSITION_4.LOWER_TOLERANCE_MINUS )
   END_RUNG
   // the same network as SCL:
   // ENO of a box is taken as its EN; it also drops when the box reports an error
   #_w1 := #MEAS_SYS_1_ACTIVE_REFERENCED OR #MEAS_SYS_2_ACTIVE_REFERENCED;
   IF #_w1 THEN
       #SAFETY_POSITION_4.POSITION_TOLERANCE_PLUS := #SAFETY_POSITION_4.HMI_POSITION + #SAFETY_POSITION_4.TOLERANCE_PLUS;
       #SAFETY_POSITION_4.POSITION_TOLERANCE_MINUS := #SAFETY_POSITION_4.HMI_POSITION - #SAFETY_POSITION_4.TOLERANCE_MINUS;
   END_IF;
   #_w2 := #_w1 AND (#SAFETY_POSITION_4.HMI_POSITION <> 1.1);
   #SAFETY_POSITION_4.IN_POSITION := #_w2 AND (#AXIS_POS >= #SAFETY_POSITION_4.POSITION_TOLERANCE_MINUS) AND (#AXIS_POS <= #SAFETY_POSITION_4.POSITION_TOLERANCE_PLUS);
   #SAFETY_POSITION_4.GREATER_TOLERANCE_PLUS := #_w2 AND (#AXIS_POS >= #SAFETY_POSITION_4.POSITION_TOLERANCE_PLUS);
   #SAFETY_POSITION_4.GREATER_TOLERANCE_MINUS := #_w2 AND (#AXIS_POS >= #SAFETY_POSITION_4.POSITION_TOLERANCE_MINUS);
   #SAFETY_POSITION_4.LOWER_TOLERANCE_PLUS := #_w2 AND (#AXIS_POS <= #SAFETY_POSITION_4.POSITION_TOLERANCE_PLUS);
   #SAFETY_POSITION_4.LOWER_TOLERANCE_MINUS := #_w2 AND (#AXIS_POS <= #SAFETY_POSITION_4.POSITION_TOLERANCE_MINUS);
END_REGION

REGION Network 12: SAFETY POSITION 5
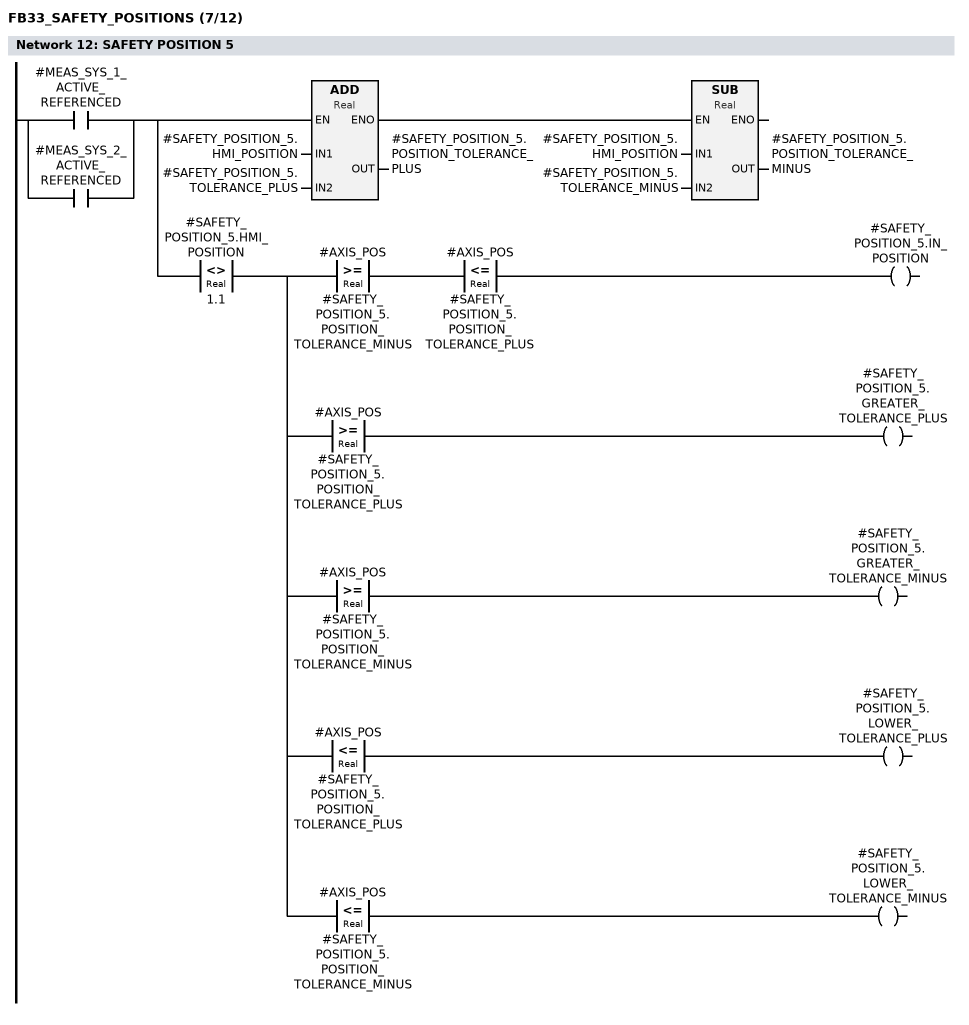
   RUNG wire#powerrail
      Contact( #MEAS_SYS_1_ACTIVE_REFERENCED )
      wire#w1
      { S7_Templates := "SrcType := Real"; S7_GenerateENO := "TRUE" } Add(in1 := #SAFETY_POSITION_5.HMI_POSITION, in2 := #SAFETY_POSITION_5.TOLERANCE_PLUS, out => #SAFETY_POSITION_5.POSITION_TOLERANCE_PLUS)
      { S7_Templates := "SrcType := Real"; S7_GenerateENO := "TRUE" } Sub(in1 := #SAFETY_POSITION_5.HMI_POSITION, in2 := #SAFETY_POSITION_5.TOLERANCE_MINUS, out => #SAFETY_POSITION_5.POSITION_TOLERANCE_MINUS)
   END_RUNG
   RUNG wire#powerrail
      Contact( #MEAS_SYS_2_ACTIVE_REFERENCED )
   END_RUNG wire#w1
   RUNG wire#w1
      { S7_Templates := "SrcType := Real" } NE_Contact(in1 := #SAFETY_POSITION_5.HMI_POSITION, in2 := 1.1)
      wire#w2
      { S7_Templates := "SrcType := Real" } GE_Contact(in1 := #AXIS_POS, in2 := #SAFETY_POSITION_5.POSITION_TOLERANCE_MINUS)
      { S7_Templates := "SrcType := Real" } LE_Contact(in1 := #AXIS_POS, in2 := #SAFETY_POSITION_5.POSITION_TOLERANCE_PLUS)
      Coil( #SAFETY_POSITION_5.IN_POSITION )
   END_RUNG
   RUNG wire#w2
      { S7_Templates := "SrcType := Real" } GE_Contact(in1 := #AXIS_POS, in2 := #SAFETY_POSITION_5.POSITION_TOLERANCE_PLUS)
      Coil( #SAFETY_POSITION_5.GREATER_TOLERANCE_PLUS )
   END_RUNG
   RUNG wire#w2
      { S7_Templates := "SrcType := Real" } GE_Contact(in1 := #AXIS_POS, in2 := #SAFETY_POSITION_5.POSITION_TOLERANCE_MINUS)
      Coil( #SAFETY_POSITION_5.GREATER_TOLERANCE_MINUS )
   END_RUNG
   RUNG wire#w2
      { S7_Templates := "SrcType := Real" } LE_Contact(in1 := #AXIS_POS, in2 := #SAFETY_POSITION_5.POSITION_TOLERANCE_PLUS)
      Coil( #SAFETY_POSITION_5.LOWER_TOLERANCE_PLUS )
   END_RUNG
   RUNG wire#w2
      { S7_Templates := "SrcType := Real" } LE_Contact(in1 := #AXIS_POS, in2 := #SAFETY_POSITION_5.POSITION_TOLERANCE_MINUS)
      Coil( #SAFETY_POSITION_5.LOWER_TOLERANCE_MINUS )
   END_RUNG
   // the same network as SCL:
   // ENO of a box is taken as its EN; it also drops when the box reports an error
   #_w1 := #MEAS_SYS_1_ACTIVE_REFERENCED OR #MEAS_SYS_2_ACTIVE_REFERENCED;
   IF #_w1 THEN
       #SAFETY_POSITION_5.POSITION_TOLERANCE_PLUS := #SAFETY_POSITION_5.HMI_POSITION + #SAFETY_POSITION_5.TOLERANCE_PLUS;
       #SAFETY_POSITION_5.POSITION_TOLERANCE_MINUS := #SAFETY_POSITION_5.HMI_POSITION - #SAFETY_POSITION_5.TOLERANCE_MINUS;
   END_IF;
   #_w2 := #_w1 AND (#SAFETY_POSITION_5.HMI_POSITION <> 1.1);
   #SAFETY_POSITION_5.IN_POSITION := #_w2 AND (#AXIS_POS >= #SAFETY_POSITION_5.POSITION_TOLERANCE_MINUS) AND (#AXIS_POS <= #SAFETY_POSITION_5.POSITION_TOLERANCE_PLUS);
   #SAFETY_POSITION_5.GREATER_TOLERANCE_PLUS := #_w2 AND (#AXIS_POS >= #SAFETY_POSITION_5.POSITION_TOLERANCE_PLUS);
   #SAFETY_POSITION_5.GREATER_TOLERANCE_MINUS := #_w2 AND (#AXIS_POS >= #SAFETY_POSITION_5.POSITION_TOLERANCE_MINUS);
   #SAFETY_POSITION_5.LOWER_TOLERANCE_PLUS := #_w2 AND (#AXIS_POS <= #SAFETY_POSITION_5.POSITION_TOLERANCE_PLUS);
   #SAFETY_POSITION_5.LOWER_TOLERANCE_MINUS := #_w2 AND (#AXIS_POS <= #SAFETY_POSITION_5.POSITION_TOLERANCE_MINUS);
END_REGION

REGION Network 13: SAFETY POSITION 6
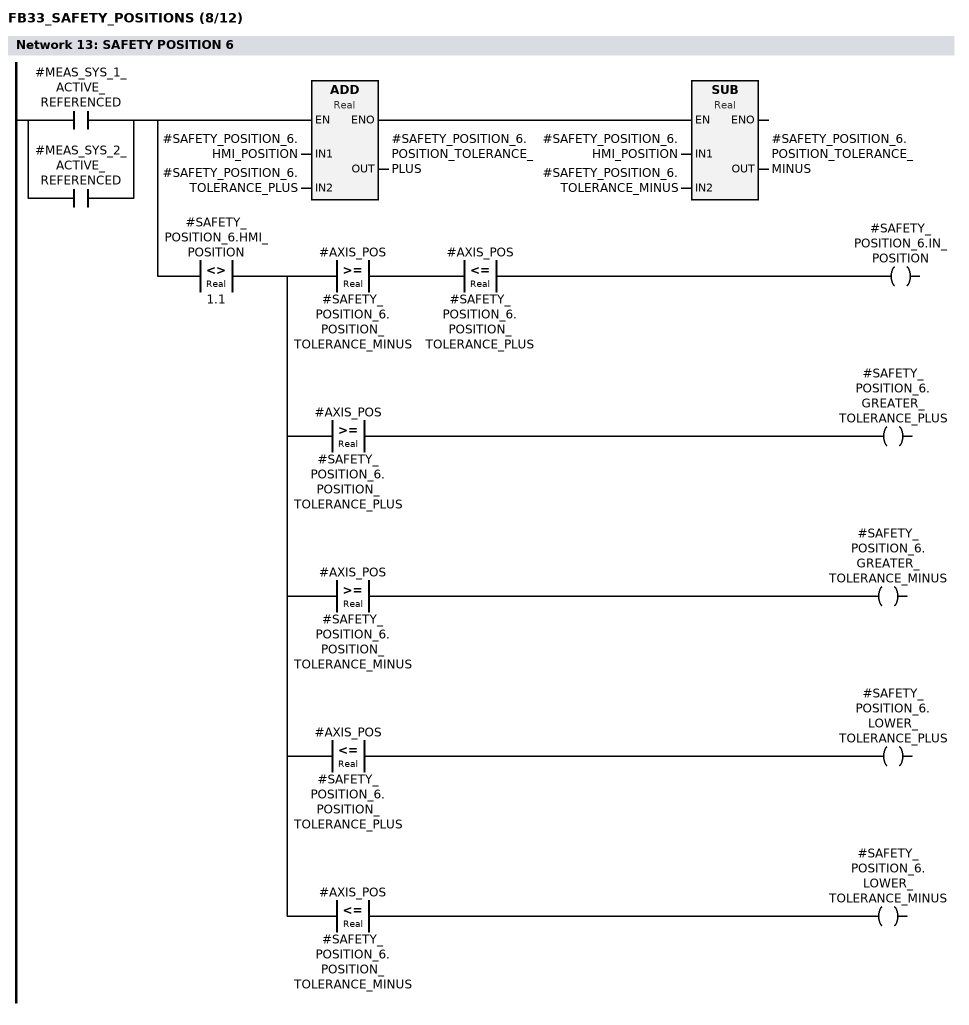
   RUNG wire#powerrail
      Contact( #MEAS_SYS_1_ACTIVE_REFERENCED )
      wire#w1
      { S7_Templates := "SrcType := Real"; S7_GenerateENO := "TRUE" } Add(in1 := #SAFETY_POSITION_6.HMI_POSITION, in2 := #SAFETY_POSITION_6.TOLERANCE_PLUS, out => #SAFETY_POSITION_6.POSITION_TOLERANCE_PLUS)
      { S7_Templates := "SrcType := Real"; S7_GenerateENO := "TRUE" } Sub(in1 := #SAFETY_POSITION_6.HMI_POSITION, in2 := #SAFETY_POSITION_6.TOLERANCE_MINUS, out => #SAFETY_POSITION_6.POSITION_TOLERANCE_MINUS)
   END_RUNG
   RUNG wire#powerrail
      Contact( #MEAS_SYS_2_ACTIVE_REFERENCED )
   END_RUNG wire#w1
   RUNG wire#w1
      { S7_Templates := "SrcType := Real" } NE_Contact(in1 := #SAFETY_POSITION_6.HMI_POSITION, in2 := 1.1)
      wire#w2
      { S7_Templates := "SrcType := Real" } GE_Contact(in1 := #AXIS_POS, in2 := #SAFETY_POSITION_6.POSITION_TOLERANCE_MINUS)
      { S7_Templates := "SrcType := Real" } LE_Contact(in1 := #AXIS_POS, in2 := #SAFETY_POSITION_6.POSITION_TOLERANCE_PLUS)
      Coil( #SAFETY_POSITION_6.IN_POSITION )
   END_RUNG
   RUNG wire#w2
      { S7_Templates := "SrcType := Real" } GE_Contact(in1 := #AXIS_POS, in2 := #SAFETY_POSITION_6.POSITION_TOLERANCE_PLUS)
      Coil( #SAFETY_POSITION_6.GREATER_TOLERANCE_PLUS )
   END_RUNG
   RUNG wire#w2
      { S7_Templates := "SrcType := Real" } GE_Contact(in1 := #AXIS_POS, in2 := #SAFETY_POSITION_6.POSITION_TOLERANCE_MINUS)
      Coil( #SAFETY_POSITION_6.GREATER_TOLERANCE_MINUS )
   END_RUNG
   RUNG wire#w2
      { S7_Templates := "SrcType := Real" } LE_Contact(in1 := #AXIS_POS, in2 := #SAFETY_POSITION_6.POSITION_TOLERANCE_PLUS)
      Coil( #SAFETY_POSITION_6.LOWER_TOLERANCE_PLUS )
   END_RUNG
   RUNG wire#w2
      { S7_Templates := "SrcType := Real" } LE_Contact(in1 := #AXIS_POS, in2 := #SAFETY_POSITION_6.POSITION_TOLERANCE_MINUS)
      Coil( #SAFETY_POSITION_6.LOWER_TOLERANCE_MINUS )
   END_RUNG
   // the same network as SCL:
   // ENO of a box is taken as its EN; it also drops when the box reports an error
   #_w1 := #MEAS_SYS_1_ACTIVE_REFERENCED OR #MEAS_SYS_2_ACTIVE_REFERENCED;
   IF #_w1 THEN
       #SAFETY_POSITION_6.POSITION_TOLERANCE_PLUS := #SAFETY_POSITION_6.HMI_POSITION + #SAFETY_POSITION_6.TOLERANCE_PLUS;
       #SAFETY_POSITION_6.POSITION_TOLERANCE_MINUS := #SAFETY_POSITION_6.HMI_POSITION - #SAFETY_POSITION_6.TOLERANCE_MINUS;
   END_IF;
   #_w2 := #_w1 AND (#SAFETY_POSITION_6.HMI_POSITION <> 1.1);
   #SAFETY_POSITION_6.IN_POSITION := #_w2 AND (#AXIS_POS >= #SAFETY_POSITION_6.POSITION_TOLERANCE_MINUS) AND (#AXIS_POS <= #SAFETY_POSITION_6.POSITION_TOLERANCE_PLUS);
   #SAFETY_POSITION_6.GREATER_TOLERANCE_PLUS := #_w2 AND (#AXIS_POS >= #SAFETY_POSITION_6.POSITION_TOLERANCE_PLUS);
   #SAFETY_POSITION_6.GREATER_TOLERANCE_MINUS := #_w2 AND (#AXIS_POS >= #SAFETY_POSITION_6.POSITION_TOLERANCE_MINUS);
   #SAFETY_POSITION_6.LOWER_TOLERANCE_PLUS := #_w2 AND (#AXIS_POS <= #SAFETY_POSITION_6.POSITION_TOLERANCE_PLUS);
   #SAFETY_POSITION_6.LOWER_TOLERANCE_MINUS := #_w2 AND (#AXIS_POS <= #SAFETY_POSITION_6.POSITION_TOLERANCE_MINUS);
END_REGION

REGION Network 14: SAFETY POSITION 7
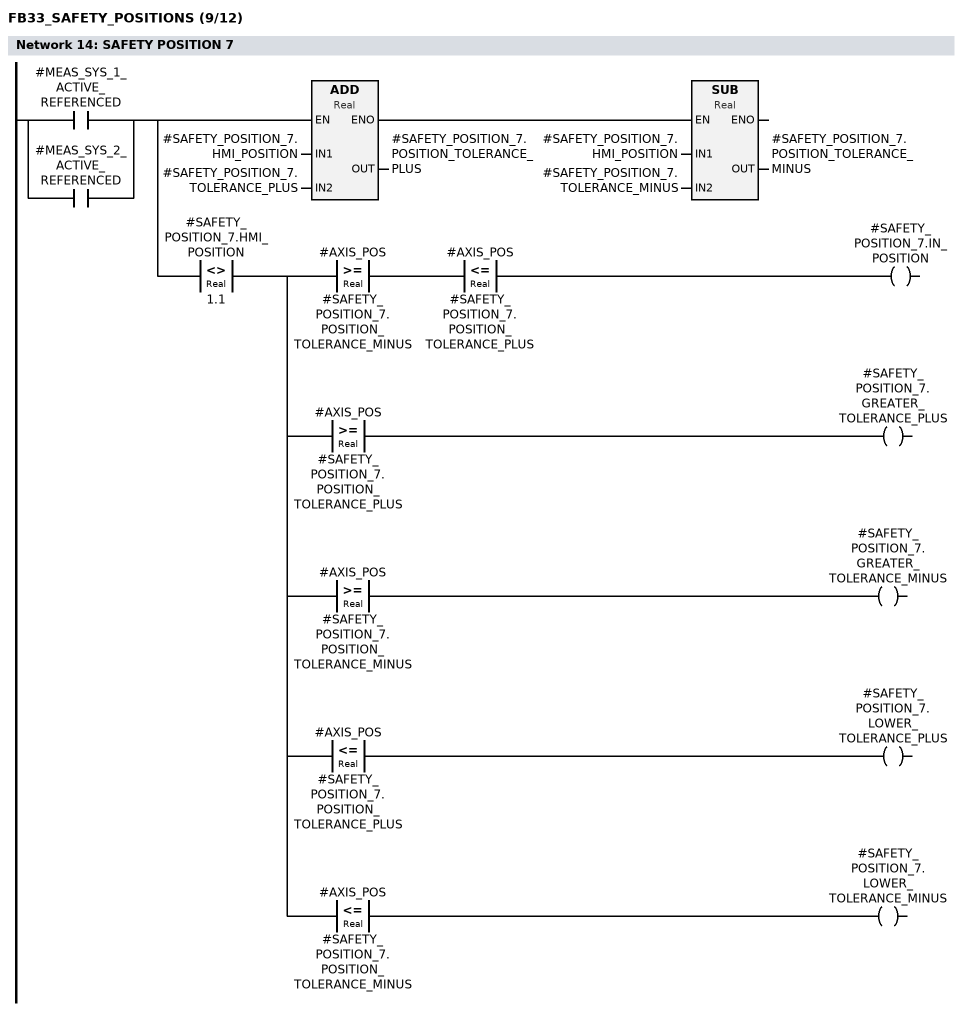
   RUNG wire#powerrail
      Contact( #MEAS_SYS_1_ACTIVE_REFERENCED )
      wire#w1
      { S7_Templates := "SrcType := Real"; S7_GenerateENO := "TRUE" } Add(in1 := #SAFETY_POSITION_7.HMI_POSITION, in2 := #SAFETY_POSITION_7.TOLERANCE_PLUS, out => #SAFETY_POSITION_7.POSITION_TOLERANCE_PLUS)
      { S7_Templates := "SrcType := Real"; S7_GenerateENO := "TRUE" } Sub(in1 := #SAFETY_POSITION_7.HMI_POSITION, in2 := #SAFETY_POSITION_7.TOLERANCE_MINUS, out => #SAFETY_POSITION_7.POSITION_TOLERANCE_MINUS)
   END_RUNG
   RUNG wire#powerrail
      Contact( #MEAS_SYS_2_ACTIVE_REFERENCED )
   END_RUNG wire#w1
   RUNG wire#w1
      { S7_Templates := "SrcType := Real" } NE_Contact(in1 := #SAFETY_POSITION_7.HMI_POSITION, in2 := 1.1)
      wire#w2
      { S7_Templates := "SrcType := Real" } GE_Contact(in1 := #AXIS_POS, in2 := #SAFETY_POSITION_7.POSITION_TOLERANCE_MINUS)
      { S7_Templates := "SrcType := Real" } LE_Contact(in1 := #AXIS_POS, in2 := #SAFETY_POSITION_7.POSITION_TOLERANCE_PLUS)
      Coil( #SAFETY_POSITION_7.IN_POSITION )
   END_RUNG
   RUNG wire#w2
      { S7_Templates := "SrcType := Real" } GE_Contact(in1 := #AXIS_POS, in2 := #SAFETY_POSITION_7.POSITION_TOLERANCE_PLUS)
      Coil( #SAFETY_POSITION_7.GREATER_TOLERANCE_PLUS )
   END_RUNG
   RUNG wire#w2
      { S7_Templates := "SrcType := Real" } GE_Contact(in1 := #AXIS_POS, in2 := #SAFETY_POSITION_7.POSITION_TOLERANCE_MINUS)
      Coil( #SAFETY_POSITION_7.GREATER_TOLERANCE_MINUS )
   END_RUNG
   RUNG wire#w2
      { S7_Templates := "SrcType := Real" } LE_Contact(in1 := #AXIS_POS, in2 := #SAFETY_POSITION_7.POSITION_TOLERANCE_PLUS)
      Coil( #SAFETY_POSITION_7.LOWER_TOLERANCE_PLUS )
   END_RUNG
   RUNG wire#w2
      { S7_Templates := "SrcType := Real" } LE_Contact(in1 := #AXIS_POS, in2 := #SAFETY_POSITION_7.POSITION_TOLERANCE_MINUS)
      Coil( #SAFETY_POSITION_7.LOWER_TOLERANCE_MINUS )
   END_RUNG
   // the same network as SCL:
   // ENO of a box is taken as its EN; it also drops when the box reports an error
   #_w1 := #MEAS_SYS_1_ACTIVE_REFERENCED OR #MEAS_SYS_2_ACTIVE_REFERENCED;
   IF #_w1 THEN
       #SAFETY_POSITION_7.POSITION_TOLERANCE_PLUS := #SAFETY_POSITION_7.HMI_POSITION + #SAFETY_POSITION_7.TOLERANCE_PLUS;
       #SAFETY_POSITION_7.POSITION_TOLERANCE_MINUS := #SAFETY_POSITION_7.HMI_POSITION - #SAFETY_POSITION_7.TOLERANCE_MINUS;
   END_IF;
   #_w2 := #_w1 AND (#SAFETY_POSITION_7.HMI_POSITION <> 1.1);
   #SAFETY_POSITION_7.IN_POSITION := #_w2 AND (#AXIS_POS >= #SAFETY_POSITION_7.POSITION_TOLERANCE_MINUS) AND (#AXIS_POS <= #SAFETY_POSITION_7.POSITION_TOLERANCE_PLUS);
   #SAFETY_POSITION_7.GREATER_TOLERANCE_PLUS := #_w2 AND (#AXIS_POS >= #SAFETY_POSITION_7.POSITION_TOLERANCE_PLUS);
   #SAFETY_POSITION_7.GREATER_TOLERANCE_MINUS := #_w2 AND (#AXIS_POS >= #SAFETY_POSITION_7.POSITION_TOLERANCE_MINUS);
   #SAFETY_POSITION_7.LOWER_TOLERANCE_PLUS := #_w2 AND (#AXIS_POS <= #SAFETY_POSITION_7.POSITION_TOLERANCE_PLUS);
   #SAFETY_POSITION_7.LOWER_TOLERANCE_MINUS := #_w2 AND (#AXIS_POS <= #SAFETY_POSITION_7.POSITION_TOLERANCE_MINUS);
END_REGION

REGION Network 15: SAFETY POSITION 8
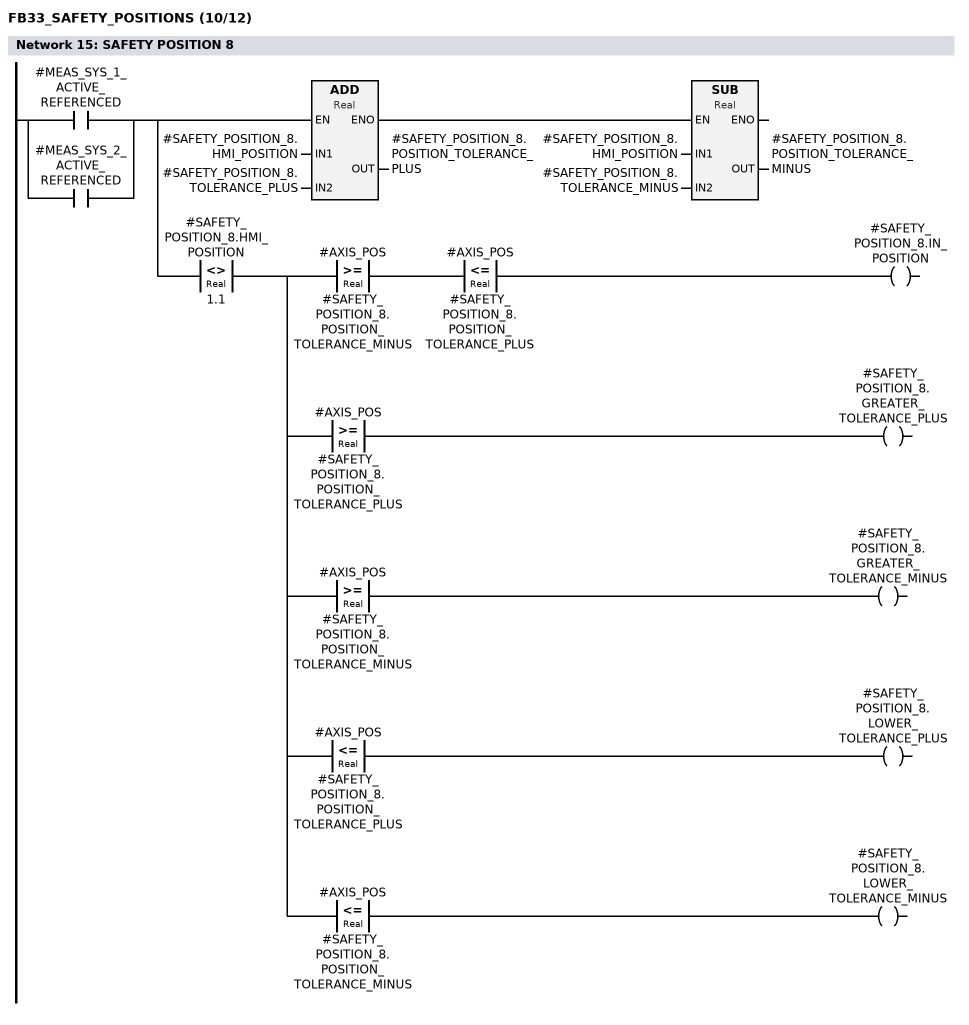
   RUNG wire#powerrail
      Contact( #MEAS_SYS_1_ACTIVE_REFERENCED )
      wire#w1
      { S7_Templates := "SrcType := Real"; S7_GenerateENO := "TRUE" } Add(in1 := #SAFETY_POSITION_8.HMI_POSITION, in2 := #SAFETY_POSITION_8.TOLERANCE_PLUS, out => #SAFETY_POSITION_8.POSITION_TOLERANCE_PLUS)
      { S7_Templates := "SrcType := Real"; S7_GenerateENO := "TRUE" } Sub(in1 := #SAFETY_POSITION_8.HMI_POSITION, in2 := #SAFETY_POSITION_8.TOLERANCE_MINUS, out => #SAFETY_POSITION_8.POSITION_TOLERANCE_MINUS)
   END_RUNG
   RUNG wire#powerrail
      Contact( #MEAS_SYS_2_ACTIVE_REFERENCED )
   END_RUNG wire#w1
   RUNG wire#w1
      { S7_Templates := "SrcType := Real" } NE_Contact(in1 := #SAFETY_POSITION_8.HMI_POSITION, in2 := 1.1)
      wire#w2
      { S7_Templates := "SrcType := Real" } GE_Contact(in1 := #AXIS_POS, in2 := #SAFETY_POSITION_8.POSITION_TOLERANCE_MINUS)
      { S7_Templates := "SrcType := Real" } LE_Contact(in1 := #AXIS_POS, in2 := #SAFETY_POSITION_8.POSITION_TOLERANCE_PLUS)
      Coil( #SAFETY_POSITION_8.IN_POSITION )
   END_RUNG
   RUNG wire#w2
      { S7_Templates := "SrcType := Real" } GE_Contact(in1 := #AXIS_POS, in2 := #SAFETY_POSITION_8.POSITION_TOLERANCE_PLUS)
      Coil( #SAFETY_POSITION_8.GREATER_TOLERANCE_PLUS )
   END_RUNG
   RUNG wire#w2
      { S7_Templates := "SrcType := Real" } GE_Contact(in1 := #AXIS_POS, in2 := #SAFETY_POSITION_8.POSITION_TOLERANCE_MINUS)
      Coil( #SAFETY_POSITION_8.GREATER_TOLERANCE_MINUS )
   END_RUNG
   RUNG wire#w2
      { S7_Templates := "SrcType := Real" } LE_Contact(in1 := #AXIS_POS, in2 := #SAFETY_POSITION_8.POSITION_TOLERANCE_PLUS)
      Coil( #SAFETY_POSITION_8.LOWER_TOLERANCE_PLUS )
   END_RUNG
   RUNG wire#w2
      { S7_Templates := "SrcType := Real" } LE_Contact(in1 := #AXIS_POS, in2 := #SAFETY_POSITION_8.POSITION_TOLERANCE_MINUS)
      Coil( #SAFETY_POSITION_8.LOWER_TOLERANCE_MINUS )
   END_RUNG
   // the same network as SCL:
   // ENO of a box is taken as its EN; it also drops when the box reports an error
   #_w1 := #MEAS_SYS_1_ACTIVE_REFERENCED OR #MEAS_SYS_2_ACTIVE_REFERENCED;
   IF #_w1 THEN
       #SAFETY_POSITION_8.POSITION_TOLERANCE_PLUS := #SAFETY_POSITION_8.HMI_POSITION + #SAFETY_POSITION_8.TOLERANCE_PLUS;
       #SAFETY_POSITION_8.POSITION_TOLERANCE_MINUS := #SAFETY_POSITION_8.HMI_POSITION - #SAFETY_POSITION_8.TOLERANCE_MINUS;
   END_IF;
   #_w2 := #_w1 AND (#SAFETY_POSITION_8.HMI_POSITION <> 1.1);
   #SAFETY_POSITION_8.IN_POSITION := #_w2 AND (#AXIS_POS >= #SAFETY_POSITION_8.POSITION_TOLERANCE_MINUS) AND (#AXIS_POS <= #SAFETY_POSITION_8.POSITION_TOLERANCE_PLUS);
   #SAFETY_POSITION_8.GREATER_TOLERANCE_PLUS := #_w2 AND (#AXIS_POS >= #SAFETY_POSITION_8.POSITION_TOLERANCE_PLUS);
   #SAFETY_POSITION_8.GREATER_TOLERANCE_MINUS := #_w2 AND (#AXIS_POS >= #SAFETY_POSITION_8.POSITION_TOLERANCE_MINUS);
   #SAFETY_POSITION_8.LOWER_TOLERANCE_PLUS := #_w2 AND (#AXIS_POS <= #SAFETY_POSITION_8.POSITION_TOLERANCE_PLUS);
   #SAFETY_POSITION_8.LOWER_TOLERANCE_MINUS := #_w2 AND (#AXIS_POS <= #SAFETY_POSITION_8.POSITION_TOLERANCE_MINUS);
END_REGION

REGION Network 16: SAFETY POSITION 9
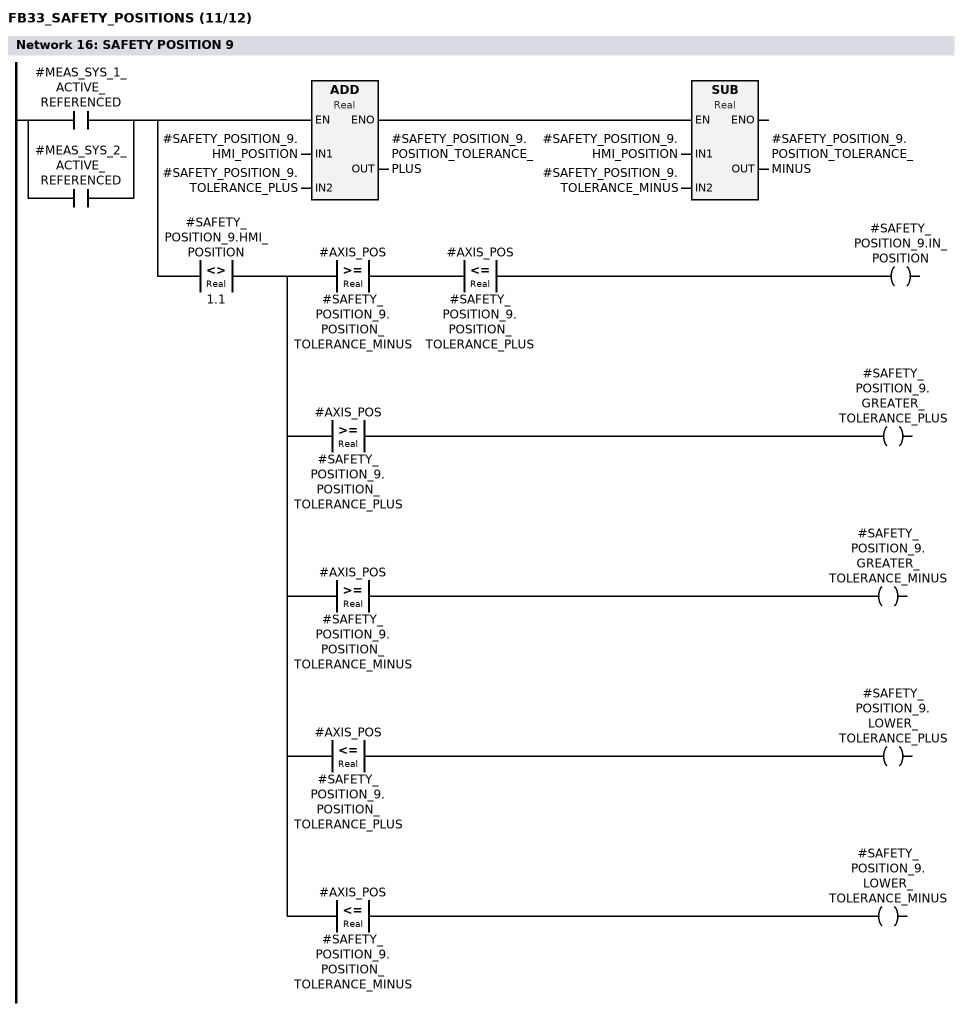
   RUNG wire#powerrail
      Contact( #MEAS_SYS_1_ACTIVE_REFERENCED )
      wire#w1
      { S7_Templates := "SrcType := Real"; S7_GenerateENO := "TRUE" } Add(in1 := #SAFETY_POSITION_9.HMI_POSITION, in2 := #SAFETY_POSITION_9.TOLERANCE_PLUS, out => #SAFETY_POSITION_9.POSITION_TOLERANCE_PLUS)
      { S7_Templates := "SrcType := Real"; S7_GenerateENO := "TRUE" } Sub(in1 := #SAFETY_POSITION_9.HMI_POSITION, in2 := #SAFETY_POSITION_9.TOLERANCE_MINUS, out => #SAFETY_POSITION_9.POSITION_TOLERANCE_MINUS)
   END_RUNG
   RUNG wire#powerrail
      Contact( #MEAS_SYS_2_ACTIVE_REFERENCED )
   END_RUNG wire#w1
   RUNG wire#w1
      { S7_Templates := "SrcType := Real" } NE_Contact(in1 := #SAFETY_POSITION_9.HMI_POSITION, in2 := 1.1)
      wire#w2
      { S7_Templates := "SrcType := Real" } GE_Contact(in1 := #AXIS_POS, in2 := #SAFETY_POSITION_9.POSITION_TOLERANCE_MINUS)
      { S7_Templates := "SrcType := Real" } LE_Contact(in1 := #AXIS_POS, in2 := #SAFETY_POSITION_9.POSITION_TOLERANCE_PLUS)
      Coil( #SAFETY_POSITION_9.IN_POSITION )
   END_RUNG
   RUNG wire#w2
      { S7_Templates := "SrcType := Real" } GE_Contact(in1 := #AXIS_POS, in2 := #SAFETY_POSITION_9.POSITION_TOLERANCE_PLUS)
      Coil( #SAFETY_POSITION_9.GREATER_TOLERANCE_PLUS )
   END_RUNG
   RUNG wire#w2
      { S7_Templates := "SrcType := Real" } GE_Contact(in1 := #AXIS_POS, in2 := #SAFETY_POSITION_9.POSITION_TOLERANCE_MINUS)
      Coil( #SAFETY_POSITION_9.GREATER_TOLERANCE_MINUS )
   END_RUNG
   RUNG wire#w2
      { S7_Templates := "SrcType := Real" } LE_Contact(in1 := #AXIS_POS, in2 := #SAFETY_POSITION_9.POSITION_TOLERANCE_PLUS)
      Coil( #SAFETY_POSITION_9.LOWER_TOLERANCE_PLUS )
   END_RUNG
   RUNG wire#w2
      { S7_Templates := "SrcType := Real" } LE_Contact(in1 := #AXIS_POS, in2 := #SAFETY_POSITION_9.POSITION_TOLERANCE_MINUS)
      Coil( #SAFETY_POSITION_9.LOWER_TOLERANCE_MINUS )
   END_RUNG
   // the same network as SCL:
   // ENO of a box is taken as its EN; it also drops when the box reports an error
   #_w1 := #MEAS_SYS_1_ACTIVE_REFERENCED OR #MEAS_SYS_2_ACTIVE_REFERENCED;
   IF #_w1 THEN
       #SAFETY_POSITION_9.POSITION_TOLERANCE_PLUS := #SAFETY_POSITION_9.HMI_POSITION + #SAFETY_POSITION_9.TOLERANCE_PLUS;
       #SAFETY_POSITION_9.POSITION_TOLERANCE_MINUS := #SAFETY_POSITION_9.HMI_POSITION - #SAFETY_POSITION_9.TOLERANCE_MINUS;
   END_IF;
   #_w2 := #_w1 AND (#SAFETY_POSITION_9.HMI_POSITION <> 1.1);
   #SAFETY_POSITION_9.IN_POSITION := #_w2 AND (#AXIS_POS >= #SAFETY_POSITION_9.POSITION_TOLERANCE_MINUS) AND (#AXIS_POS <= #SAFETY_POSITION_9.POSITION_TOLERANCE_PLUS);
   #SAFETY_POSITION_9.GREATER_TOLERANCE_PLUS := #_w2 AND (#AXIS_POS >= #SAFETY_POSITION_9.POSITION_TOLERANCE_PLUS);
   #SAFETY_POSITION_9.GREATER_TOLERANCE_MINUS := #_w2 AND (#AXIS_POS >= #SAFETY_POSITION_9.POSITION_TOLERANCE_MINUS);
   #SAFETY_POSITION_9.LOWER_TOLERANCE_PLUS := #_w2 AND (#AXIS_POS <= #SAFETY_POSITION_9.POSITION_TOLERANCE_PLUS);
   #SAFETY_POSITION_9.LOWER_TOLERANCE_MINUS := #_w2 AND (#AXIS_POS <= #SAFETY_POSITION_9.POSITION_TOLERANCE_MINUS);
END_REGION

REGION Network 17: SAFETY POSITION 10
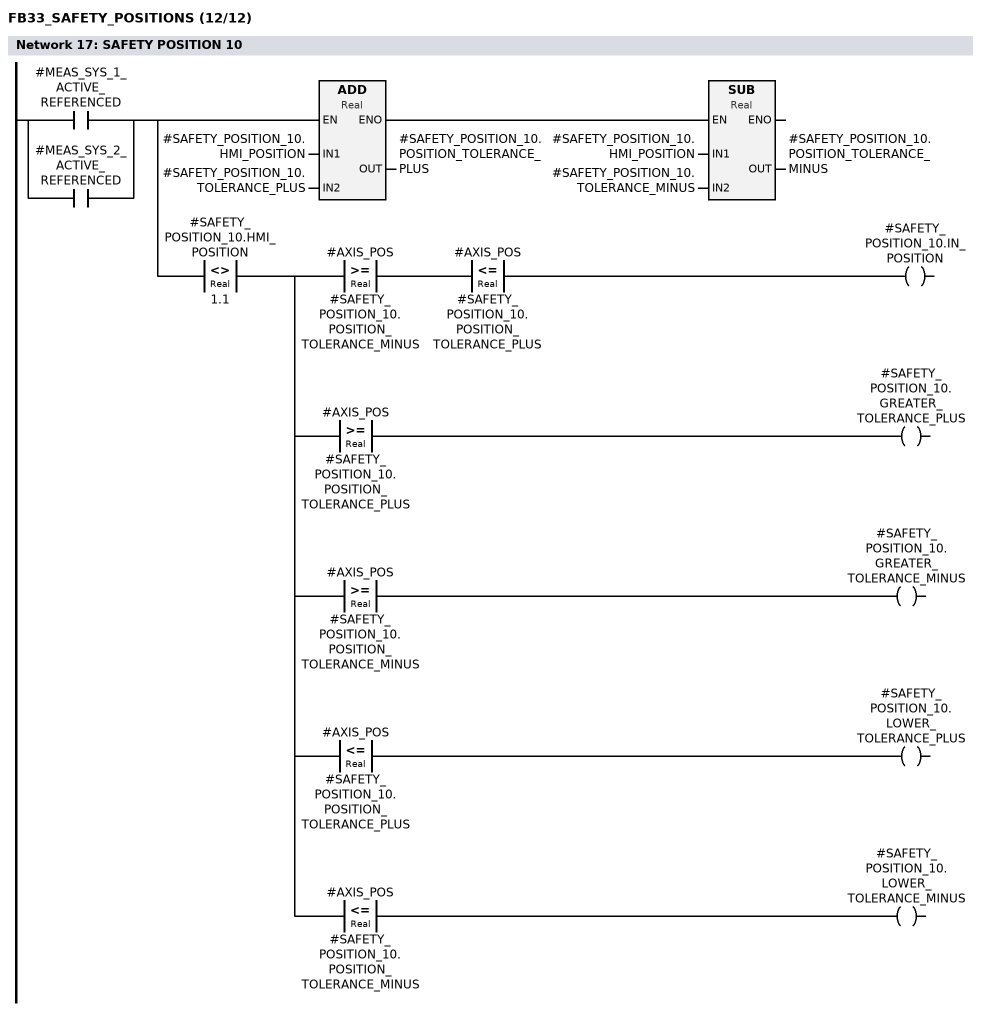
   RUNG wire#powerrail
      Contact( #MEAS_SYS_1_ACTIVE_REFERENCED )
      wire#w1
      { S7_Templates := "SrcType := Real"; S7_GenerateENO := "TRUE" } Add(in1 := #SAFETY_POSITION_10.HMI_POSITION, in2 := #SAFETY_POSITION_10.TOLERANCE_PLUS, out => #SAFETY_POSITION_10.POSITION_TOLERANCE_PLUS)
      { S7_Templates := "SrcType := Real"; S7_GenerateENO := "TRUE" } Sub(in1 := #SAFETY_POSITION_10.HMI_POSITION, in2 := #SAFETY_POSITION_10.TOLERANCE_MINUS, out => #SAFETY_POSITION_10.POSITION_TOLERANCE_MINUS)
   END_RUNG
   RUNG wire#powerrail
      Contact( #MEAS_SYS_2_ACTIVE_REFERENCED )
   END_RUNG wire#w1
   RUNG wire#w1
      { S7_Templates := "SrcType := Real" } NE_Contact(in1 := #SAFETY_POSITION_10.HMI_POSITION, in2 := 1.1)
      wire#w2
      { S7_Templates := "SrcType := Real" } GE_Contact(in1 := #AXIS_POS, in2 := #SAFETY_POSITION_10.POSITION_TOLERANCE_MINUS)
      { S7_Templates := "SrcType := Real" } LE_Contact(in1 := #AXIS_POS, in2 := #SAFETY_POSITION_10.POSITION_TOLERANCE_PLUS)
      Coil( #SAFETY_POSITION_10.IN_POSITION )
   END_RUNG
   RUNG wire#w2
      { S7_Templates := "SrcType := Real" } GE_Contact(in1 := #AXIS_POS, in2 := #SAFETY_POSITION_10.POSITION_TOLERANCE_PLUS)
      Coil( #SAFETY_POSITION_10.GREATER_TOLERANCE_PLUS )
   END_RUNG
   RUNG wire#w2
      { S7_Templates := "SrcType := Real" } GE_Contact(in1 := #AXIS_POS, in2 := #SAFETY_POSITION_10.POSITION_TOLERANCE_MINUS)
      Coil( #SAFETY_POSITION_10.GREATER_TOLERANCE_MINUS )
   END_RUNG
   RUNG wire#w2
      { S7_Templates := "SrcType := Real" } LE_Contact(in1 := #AXIS_POS, in2 := #SAFETY_POSITION_10.POSITION_TOLERANCE_PLUS)
      Coil( #SAFETY_POSITION_10.LOWER_TOLERANCE_PLUS )
   END_RUNG
   RUNG wire#w2
      { S7_Templates := "SrcType := Real" } LE_Contact(in1 := #AXIS_POS, in2 := #SAFETY_POSITION_10.POSITION_TOLERANCE_MINUS)
      Coil( #SAFETY_POSITION_10.LOWER_TOLERANCE_MINUS )
   END_RUNG
   // the same network as SCL:
   // ENO of a box is taken as its EN; it also drops when the box reports an error
   #_w1 := #MEAS_SYS_1_ACTIVE_REFERENCED OR #MEAS_SYS_2_ACTIVE_REFERENCED;
   IF #_w1 THEN
       #SAFETY_POSITION_10.POSITION_TOLERANCE_PLUS := #SAFETY_POSITION_10.HMI_POSITION + #SAFETY_POSITION_10.TOLERANCE_PLUS;
       #SAFETY_POSITION_10.POSITION_TOLERANCE_MINUS := #SAFETY_POSITION_10.HMI_POSITION - #SAFETY_POSITION_10.TOLERANCE_MINUS;
   END_IF;
   #_w2 := #_w1 AND (#SAFETY_POSITION_10.HMI_POSITION <> 1.1);
   #SAFETY_POSITION_10.IN_POSITION := #_w2 AND (#AXIS_POS >= #SAFETY_POSITION_10.POSITION_TOLERANCE_MINUS) AND (#AXIS_POS <= #SAFETY_POSITION_10.POSITION_TOLERANCE_PLUS);
   #SAFETY_POSITION_10.GREATER_TOLERANCE_PLUS := #_w2 AND (#AXIS_POS >= #SAFETY_POSITION_10.POSITION_TOLERANCE_PLUS);
   #SAFETY_POSITION_10.GREATER_TOLERANCE_MINUS := #_w2 AND (#AXIS_POS >= #SAFETY_POSITION_10.POSITION_TOLERANCE_MINUS);
   #SAFETY_POSITION_10.LOWER_TOLERANCE_PLUS := #_w2 AND (#AXIS_POS <= #SAFETY_POSITION_10.POSITION_TOLERANCE_PLUS);
   #SAFETY_POSITION_10.LOWER_TOLERANCE_MINUS := #_w2 AND (#AXIS_POS <= #SAFETY_POSITION_10.POSITION_TOLERANCE_MINUS);
END_REGION
END_FUNCTION_BLOCK
